(* CODESYS project mobject-datatypes.library
   Company: mobject
   DefaultNamespace: mobject-datatypes
   Version: 0.7.0
   Placeholder: mobject-datatypes
   Author: mobject dev team
   Title: mobject-datatypes

Project tree, tasks and I/O mapping:
  libraries: mobject-collections, 1.2.0 (mobject); mobject-constants-datatype-limits, 1.0.0 (mobject); mobject-deserialization, 0.2.0 (mobject); mobject-disposable, 1.0.0 (mobject); mobject-enumerable, 1.1.0 (mobject); mobject-errors, 0.2.0 (mobject); mobject-events, 1.0.0 (mobject); mobject-serialization, 0.4.0 (mobject); Tc2_Standard, * (Beckhoff Automation GmbH); Tc2_System, * (Beckhoff Automation GmbH); Tc2_Utilities, * (Beckhoff Automation GmbH)
  _Internal/
    Datatype/
      function block DatatypeBase [ST]: OnSerializeTypeWith, Accept, Address, ClearReference, Clone, IsUserDefined, SerializeTypeWith, SerializeWith, Size, TryCopyFrom, TryDeserializeFrom, TryMakeReferenceTo, TryResolveAsAliasDatatype, TryResolveAsEnumDatatype, TryResolveAsInterfaceDatatype, TryResolveAsStructuredDatatype, TypeName
    Errors/
      function block UnknownEnumerationError [ST]: FB_init, ErrorType, Message
    Events/
      function block AliasDatatypeAddedEvent [ST]: FB_init, Target
      function block DatatypeAddedEvent [ST]: FB_init, Target
      function block EnumDatatypeAddedEvent [ST]: FB_init, Target
      function block StructuredDatatypeAddedEvent [ST]: FB_init, Target
    StructureMembers/
      Host/
        function block StructureMemberHost [ST]: Accept, AddMember, GetMemberEnumerator, SerializeTypeWith, SerializeWith, TryDeserializeFrom, TryGetMemberByName
      Interface/
        interface I_HostStructureMembers: Members
        interface I_StructureMembers: Accept, GetMemberEnumerator, TryGetMemberByName
  Datatype/
    Interface/
      interface I_AliasDatatype: BaseDatatype
      interface I_Datatype: Accept, Address, ClearReference, Clone, IsUserDefined, SerializeTypeWith, Size, TryCopyFrom, TryDeserializeFrom, TryMakeReferenceTo, TryResolveAsAliasDatatype, TryResolveAsEnumDatatype, TryResolveAsInterfaceDatatype, TryResolveAsStructuredDatatype, TypeName
      interface I_EnumDatatype
      interface I_InterfaceDatatype: Identifier
      interface I_NumericDatatype: IsFloat, IsSigned
      interface I_StructuredDatatype
      interface I_UserDefinedDatatype: Identifier
    function block AliasDatatypeBase [ST]: AddBaseDatatype, OnSerializeTypeWith, BaseDatatype, SerializeWith, TryDeserializeFrom, TryResolveAsAliasDatatype, TypeName
    function block EnumDatatypeBase [ST]: CreateEnumError, SerializeBaseType, SerializeEnums, AddBaseDatatype, AddEnumeration, IsEnumeratorValueEqual, OnSerializeTypeWith, BaseDatatype, SerializeWith, TryDeserializeFrom, TryResolveAsEnumDatatype, TypeName
    function block InterfaceDatatypeBase [ST]: OnSerializeTypeWith, Identifier, IsUserDefined, TryCopyFrom, TryResolveAsInterfaceDatatype, TypeName
    function block NumericDatatypeBase [ST]: OnSerializeTypeWith, SerializeMaxValue, SerializeMinValue, IsFloat, IsSigned
    function block StructuredDatatypeBase [ST]: AddMember, OnSerializeTypeWith, Accept, Members, SerializeWith, TryDeserializeFrom, TryResolveAsStructuredDatatype, TypeName
    function block UserDefinedDatatypeBase [ST]: OnSerializeTypeWith, Identifier, IsUserDefined, TryCopyFrom
  DatatypeOperations/
    Collection/
      function block DatatypeOperations [ST]: FB_exit, CreateMemoryCopyOperation, CreateSafeMemoryCopyOperation, AddMemoryCopyOperation, AddSafeMemoryCopyOperation, Clear, Execute
    Interface/
      interface I_DatatypeOperation: Execute
    function block MemCopyOperation [ST]: FB_init, Execute
    function block SafeMemCopyOperation [ST]: FB_init, Execute
  DatatypePack/
    interface I_DatatypePack: RegisterWith
  Datatypes/
    Base/
      function block Datatypes [ST]: AcceptAlias, AcceptEnum, AcceptPrimative, AcceptStructures, SerializeAliasTypeWith, SerializeEnumsTypeWith, SerializePrimitiveTypeWith, SerializeStructuresTypeWith, EmitOnAliasDatatypeAddedEvent, EmitOnDatatypeAddedEvent, EmitOnEnumDatatypeAddedEvent, EmitOnStructuredDatatypeAddedEvent, Accept, GetAliasByIdentifier, GetEnumByIdentifier, GetPrimitiveByTypeName, GetStructureByIdentifier, OffEvent, OnceEvent, OnEvent, RegisterDatatype, SerializeTypeWith
    Events/
      interface I_AliasDatatypeAddedEvent: Target
      interface I_DatatypeAddedEvent: Target
      interface I_EnumDatatypeAddedEvent: Target
      interface I_StructuredDatatypeAddedEvent: Target
    Interface/
      interface I_Datatypes: Accept, GetAliasByIdentifier, GetPrimitiveByTypeName, GetStructureByIdentifier, RegisterDatatype, SerializeTypeWith
  DatatypeVisitor/
    interface I_DatatypeVisitor: VisitDatatype
  Primitive/
    function block _BOOL [ST]: FB_init, Address, ClearReference, Clone, MakeReferenceTo, SerializeWith, Size, TryDeserializeFrom, TryMakeReferenceTo, TypeName, Value
    function block _BYTE [ST]: FB_init, SerializeMaxValue, SerializeMinValue, Address, ClearReference, Clone, IsFloat, IsSigned, MakeReferenceTo, MaxValue, MinValue, SerializeWith, Size, TryDeserializeFrom, TryMakeReferenceTo, TypeName, Value
    function block _DINT [ST]: FB_init, SerializeMaxValue, SerializeMinValue, Address, ClearReference, Clone, IsFloat, IsSigned, MakeReferenceTo, MaxValue, MinValue, SerializeWith, Size, TryDeserializeFrom, TryMakeReferenceTo, TypeName, Value
    function block _DT [ST]: FB_init, Address, ClearReference, Clone, MakeReferenceTo, SerializeWith, Size, TryDeserializeFrom, TryMakeReferenceTo, TypeName, Value
    function block _DWORD [ST]: FB_init, SerializeMaxValue, SerializeMinValue, Address, ClearReference, Clone, IsFloat, IsSigned, MakeReferenceTo, MaxValue, MinValue, SerializeWith, Size, TryDeserializeFrom, TryMakeReferenceTo, TypeName, Value
    function block _INT [ST]: FB_init, SerializeMaxValue, SerializeMinValue, Address, ClearReference, Clone, IsFloat, IsSigned, MakeReferenceTo, MaxValue, MinValue, SerializeWith, Size, TryDeserializeFrom, TryMakeReferenceTo, TypeName, Value
    function block _LINT [ST]: FB_init, SerializeMaxValue, SerializeMinValue, Address, ClearReference, Clone, IsFloat, IsSigned, MakeReferenceTo, MaxValue, MinValue, SerializeWith, Size, TryDeserializeFrom, TryMakeReferenceTo, TypeName, Value
    function block _LREAL [ST]: FB_init, SerializeMaxValue, SerializeMinValue, Address, ClearReference, Clone, IsFloat, IsSigned, MakeReferenceTo, MaxValue, MinValue, SerializeWith, Size, TryDeserializeFrom, TryMakeReferenceTo, TypeName, Value
    function block _LWORD [ST]: FB_init, SerializeMaxValue, SerializeMinValue, Address, ClearReference, Clone, IsFloat, IsSigned, MakeReferenceTo, MaxValue, MinValue, SerializeWith, Size, TryDeserializeFrom, TryMakeReferenceTo, TypeName, Value
    function block _REAL [ST]: FB_init, SerializeMaxValue, SerializeMinValue, Address, ClearReference, Clone, IsFloat, IsSigned, MakeReferenceTo, MaxValue, MinValue, SerializeWith, Size, TryDeserializeFrom, TryMakeReferenceTo, TypeName, Value
    function block _SINT [ST]: FB_init, SerializeMaxValue, SerializeMinValue, Address, ClearReference, Clone, IsFloat, IsSigned, MakeReferenceTo, MaxValue, MinValue, SerializeWith, Size, TryDeserializeFrom, TryMakeReferenceTo, TypeName, Value
    function block _STRING [ST]: FB_init, Address, ClearReference, Clone, MakeReferenceTo, SerializeWith, Size, TryDeserializeFrom, TryMakeReferenceTo, TypeName, Value
    function block _TIME_OF_DAY [ST]: FB_init, Address, ClearReference, Clone, MakeReferenceTo, SerializeWith, Size, TryDeserializeFrom, TryMakeReferenceTo, TypeName, Value
    function block _TOD [ST]: FB_init, Address, ClearReference, Clone, MakeReferenceTo, SerializeWith, Size, TryDeserializeFrom, TryMakeReferenceTo, TypeName, Value
    function block _UDINT [ST]: FB_init, SerializeMaxValue, SerializeMinValue, Address, ClearReference, Clone, IsFloat, IsSigned, MakeReferenceTo, MaxValue, MinValue, SerializeWith, Size, TryDeserializeFrom, TryMakeReferenceTo, TypeName, Value
    function block _UINT [ST]: FB_init, SerializeMaxValue, SerializeMinValue, Address, ClearReference, Clone, IsFloat, IsSigned, MakeReferenceTo, MaxValue, MinValue, SerializeWith, Size, TryDeserializeFrom, TryMakeReferenceTo, TypeName, Value
    function block _ULINT [ST]: FB_init, SerializeMaxValue, SerializeMinValue, Address, ClearReference, Clone, IsFloat, IsSigned, MakeReferenceTo, MaxValue, MinValue, SerializeWith, Size, TryDeserializeFrom, TryMakeReferenceTo, TypeName, Value
    function block _USINT [ST]: FB_init, SerializeMaxValue, SerializeMinValue, Address, ClearReference, Clone, IsFloat, IsSigned, MakeReferenceTo, MaxValue, MinValue, SerializeWith, Size, TryDeserializeFrom, TryMakeReferenceTo, TypeName, Value
    function block _WORD [ST]: FB_init, SerializeMaxValue, SerializeMinValue, Address, ClearReference, Clone, IsFloat, IsSigned, MakeReferenceTo, MaxValue, MinValue, SerializeWith, Size, TryDeserializeFrom, TryMakeReferenceTo, TypeName, Value
  function block PrimitiveDatatypePack [ST]: RegisterWith
*)

// _Internal/Datatype/DatatypeBase
{attribute 'linkalways'} 
{attribute 'no_explicit_call' := 'This FB is a CLASS and must be accessed using methods or properties'}
{attribute 'enable_dynamic_creation'}
FUNCTION_BLOCK ABSTRACT DatatypeBase EXTENDS Disposable IMPLEMENTS I_Datatype
VAR
END_VAR

METHOD PROTECTED OnSerializeTypeWith
VAR_INPUT
	Serializer : I_Serializer;
END_VAR
Serializer.AddKeyString('typeName',TypeName);
END_METHOD

METHOD PUBLIC Accept
VAR_INPUT
	Visitor : I_DatatypeVisitor;
END_VAR
Visitor.VisitDatatype(this^);
END_METHOD

PROPERTY PUBLIC ABSTRACT Address : PVOID
GET
END_GET
END_PROPERTY

METHOD PUBLIC ABSTRACT ClearReference
VAR_INPUT
END_VAR
END_METHOD

METHOD PUBLIC ABSTRACT Clone : I_Datatype
END_METHOD

PROPERTY PUBLIC IsUserDefined : BOOL
GET
IsUserDefined := FALSE;
END_GET
END_PROPERTY

METHOD PUBLIC SerializeTypeWith
VAR_INPUT
	Serializer : I_Serializer;
END_VAR
Serializer.StartObject();
OnSerializeTypeWith(Serializer);
Serializer.EndObject();
END_METHOD

METHOD PUBLIC ABSTRACT SerializeWith
VAR_INPUT
	Serializer : I_Serializer;
END_VAR
END_METHOD

PROPERTY PUBLIC ABSTRACT Size : UDINT
GET
END_GET
END_PROPERTY

METHOD PUBLIC TryCopyFrom : BOOL
VAR_INPUT
	Source : I_Datatype;
END_VAR
IF Source.TypeName <> TypeName THEN
	RETURN;
END_IF

memcpy(Address, Source.Address, Size);
TryCopyFrom := TRUE;
END_METHOD

METHOD PUBLIC ABSTRACT TryDeserializeFrom : BOOL
VAR_INPUT
	Deserializer : I_Deserializer;
	Feedback : I_DeserializerFeedback;
END_VAR
END_METHOD

METHOD PUBLIC ABSTRACT TryMakeReferenceTo : BOOL
VAR_INPUT
	Target : I_Datatype;
END_VAR
END_METHOD

METHOD PUBLIC TryResolveAsAliasDatatype : BOOL
VAR_INPUT
	Destination : REFERENCE TO I_AliasDatatype;
END_VAR
TryResolveAsAliasDatatype := FALSE;
END_METHOD

METHOD PUBLIC TryResolveAsEnumDatatype : BOOL
VAR_INPUT
	Destination : REFERENCE TO I_EnumDatatype;
END_VAR
TryResolveAsEnumDatatype := FALSE;
END_METHOD

METHOD PUBLIC TryResolveAsInterfaceDatatype : BOOL
VAR_INPUT
	Destination : REFERENCE TO I_InterfaceDatatype;
END_VAR
TryResolveAsInterfaceDatatype := FALSE;
END_METHOD

METHOD PUBLIC TryResolveAsStructuredDatatype : BOOL
VAR_INPUT
	Destination : REFERENCE TO I_StructuredDatatype;
END_VAR
TryResolveAsStructuredDatatype := FALSE;
END_METHOD

PROPERTY PUBLIC ABSTRACT TypeName : T_MAXSTRING
GET
END_GET
END_PROPERTY

END_FUNCTION_BLOCK

// Datatype/Interface/I_Datatype
INTERFACE I_Datatype extends I_Serializable, I_Deserializable, I_Disposable

METHOD PUBLIC Accept
VAR_INPUT
	Visitor : I_DatatypeVisitor;
END_VAR
END_METHOD

PROPERTY PUBLIC Address : PVOID
GET
END_GET
END_PROPERTY

METHOD PUBLIC ClearReference
VAR_INPUT
END_VAR
END_METHOD

METHOD Clone : I_Datatype
END_METHOD

PROPERTY PUBLIC IsUserDefined : BOOL
GET
END_GET
END_PROPERTY

METHOD PUBLIC SerializeTypeWith
VAR_INPUT
	Serializer : I_Serializer;
END_VAR
END_METHOD

PROPERTY PUBLIC Size : UDINT
GET
END_GET
END_PROPERTY

METHOD PUBLIC TryCopyFrom : BOOL
VAR_INPUT
	Source : I_Datatype;
END_VAR
END_METHOD

METHOD PUBLIC ABSTRACT TryDeserializeFrom : BOOL
VAR_INPUT
	Deserializer : I_Deserializer;
	Feedback : I_DeserializerFeedback;
END_VAR
END_METHOD

METHOD TryMakeReferenceTo : BOOL
VAR_INPUT
	Target : I_Datatype;
END_VAR
END_METHOD

METHOD PUBLIC TryResolveAsAliasDatatype : BOOL
VAR_INPUT
	Destination : REFERENCE TO I_AliasDatatype;
END_VAR
END_METHOD

METHOD PUBLIC TryResolveAsEnumDatatype : BOOL
VAR_INPUT
	Destination : REFERENCE TO I_EnumDatatype;
END_VAR
END_METHOD

METHOD PUBLIC TryResolveAsInterfaceDatatype : BOOL
VAR_INPUT
	Destination : REFERENCE TO I_InterfaceDatatype;
END_VAR
END_METHOD

METHOD PUBLIC TryResolveAsStructuredDatatype : BOOL
VAR_INPUT
	Destination : REFERENCE TO I_StructuredDatatype;
END_VAR
END_METHOD

PROPERTY PUBLIC TypeName : T_MAXSTRING
GET
END_GET
END_PROPERTY

END_INTERFACE

// DatatypeVisitor/I_DatatypeVisitor
INTERFACE I_DatatypeVisitor

METHOD VisitDatatype
VAR_INPUT
	VisitingDatatype : I_Datatype;
END_VAR
END_METHOD

END_INTERFACE

// Datatype/Interface/I_AliasDatatype
INTERFACE I_AliasDatatype EXTENDS I_UserDefinedDatatype

PROPERTY PUBLIC BaseDatatype : I_Datatype
GET
END_GET
END_PROPERTY

END_INTERFACE

// Datatype/Interface/I_UserDefinedDatatype
INTERFACE I_UserDefinedDatatype EXTENDS I_Datatype

PROPERTY PUBLIC Identifier : T_MAXSTRING
GET
END_GET
END_PROPERTY

END_INTERFACE

// Datatype/Interface/I_EnumDatatype
INTERFACE I_EnumDatatype EXTENDS I_UserDefinedDatatype

END_INTERFACE

// Datatype/Interface/I_InterfaceDatatype
INTERFACE I_InterfaceDatatype EXTENDS I_Datatype

PROPERTY PUBLIC Identifier : T_MAXSTRING
GET
END_GET
END_PROPERTY

END_INTERFACE

// Datatype/Interface/I_StructuredDatatype
INTERFACE I_StructuredDatatype EXTENDS I_UserDefinedDatatype, I_HostStructureMembers

END_INTERFACE

// _Internal/StructureMembers/Interface/I_HostStructureMembers
INTERFACE I_HostStructureMembers EXTENDS __SYSTEM.IQueryInterface

PROPERTY PUBLIC Members : I_StructureMembers
GET
END_GET
END_PROPERTY

END_INTERFACE

// _Internal/StructureMembers/Interface/I_StructureMembers
INTERFACE I_StructureMembers

METHOD PUBLIC Accept
VAR_INPUT
	Visitor : I_DatatypeVisitor;
END_VAR
END_METHOD

METHOD PUBLIC GetMemberEnumerator : I_KeyValueForwardEnumerator
VAR_INPUT
END_VAR
END_METHOD

METHOD PUBLIC TryGetMemberByName : BOOL
VAR_INPUT
	Name : T_MAXSTRING;
	Destination : REFERENCE TO I_Datatype;
END_VAR
END_METHOD

END_INTERFACE

// _Internal/Errors/UnknownEnumerationError
{attribute 'linkalways'} 
{attribute 'no_explicit_call' := 'This FB is a CLASS and must be accessed using methods or properties'}
{attribute 'enable_dynamic_creation'}
FUNCTION_BLOCK UnknownEnumerationError EXTENDS Error
VAR
	enumString : T_MAXSTRING;
END_VAR

METHOD FB_init : BOOL
VAR_INPUT
	bInitRetains : BOOL; // if TRUE, the retain variables are initialized (warm start / cold start)
	bInCopyCode : BOOL;  // if TRUE, the instance afterwards gets moved into the copy code (online change)
	EnumString : T_MAXSTRING;
END_VAR
THIS^.enumString := EnumString;
END_METHOD

PROPERTY PUBLIC ErrorType : T_MAXSTRING
GET
ErrorType := 'UNKNOWN_ENUMERATION_ERROR';
END_GET
END_PROPERTY

PROPERTY PUBLIC Message : T_MAXSTRING
GET
Message := CONCAT('Unknown Enumeration : ', enumString);
END_GET
END_PROPERTY

END_FUNCTION_BLOCK

// _Internal/Events/AliasDatatypeAddedEvent
{attribute 'linkalways'} 
{attribute 'no_explicit_call' := 'This FB is a CLASS and must be accessed using methods or properties'}
{attribute 'enable_dynamic_creation'}
FUNCTION_BLOCK AliasDatatypeAddedEvent EXTENDS Disposable IMPLEMENTS I_AliasDatatypeAddedEvent
VAR
	_target : I_AliasDatatype;
END_VAR

METHOD FB_init : BOOL
VAR_INPUT
	bInitRetains : BOOL; // if TRUE, the retain variables are initialized (warm start / cold start)
	bInCopyCode : BOOL;  // if TRUE, the instance afterwards gets moved into the copy code (online change)
	Target : I_AliasDatatype;
END_VAR
This^._target := Target;
END_METHOD

PROPERTY PUBLIC Target : I_AliasDatatype
GET
Target := _target;
END_GET
END_PROPERTY

END_FUNCTION_BLOCK

// Datatypes/Events/I_AliasDatatypeAddedEvent
INTERFACE I_AliasDatatypeAddedEvent EXTENDS I_Event

PROPERTY PUBLIC Target : I_AliasDatatype
GET
END_GET
END_PROPERTY

END_INTERFACE

// _Internal/Events/DatatypeAddedEvent
{attribute 'linkalways'} 
{attribute 'no_explicit_call' := 'This FB is a CLASS and must be accessed using methods or properties'}
{attribute 'enable_dynamic_creation'}
FUNCTION_BLOCK DatatypeAddedEvent EXTENDS Disposable IMPLEMENTS I_DatatypeAddedEvent
VAR
	_target : I_Datatype;
END_VAR

METHOD FB_init : BOOL
VAR_INPUT
	bInitRetains : BOOL; // if TRUE, the retain variables are initialized (warm start / cold start)
	bInCopyCode : BOOL;  // if TRUE, the instance afterwards gets moved into the copy code (online change)
	Target : I_Datatype;
END_VAR
This^._target := Target;
END_METHOD

PROPERTY PUBLIC Target : I_Datatype
GET
Target := _target;
END_GET
END_PROPERTY

END_FUNCTION_BLOCK

// Datatypes/Events/I_DatatypeAddedEvent
INTERFACE I_DatatypeAddedEvent EXTENDS I_Event

PROPERTY PUBLIC Target : I_Datatype
GET
END_GET
END_PROPERTY

END_INTERFACE

// _Internal/Events/EnumDatatypeAddedEvent
{attribute 'linkalways'} 
{attribute 'no_explicit_call' := 'This FB is a CLASS and must be accessed using methods or properties'}
{attribute 'enable_dynamic_creation'}
FUNCTION_BLOCK EnumDatatypeAddedEvent EXTENDS Disposable IMPLEMENTS I_EnumDatatypeAddedEvent
VAR
	_target : I_EnumDatatype;
END_VAR

METHOD FB_init : BOOL
VAR_INPUT
	bInitRetains : BOOL; // if TRUE, the retain variables are initialized (warm start / cold start)
	bInCopyCode : BOOL;  // if TRUE, the instance afterwards gets moved into the copy code (online change)
	Target : I_EnumDatatype;
END_VAR
This^._target := Target;
END_METHOD

PROPERTY PUBLIC Target : I_EnumDatatype
GET
Target := _target;
END_GET
END_PROPERTY

END_FUNCTION_BLOCK

// Datatypes/Events/I_EnumDatatypeAddedEvent
INTERFACE I_EnumDatatypeAddedEvent EXTENDS I_Event

PROPERTY PUBLIC Target : I_EnumDatatype
GET
END_GET
END_PROPERTY

END_INTERFACE

// _Internal/Events/StructuredDatatypeAddedEvent
{attribute 'linkalways'} 
{attribute 'no_explicit_call' := 'This FB is a CLASS and must be accessed using methods or properties'}
{attribute 'enable_dynamic_creation'}
FUNCTION_BLOCK StructuredDatatypeAddedEvent EXTENDS Disposable IMPLEMENTS I_StructuredDatatypeAddedEvent
VAR
	_target : I_StructuredDatatype;
END_VAR

METHOD FB_init : BOOL
VAR_INPUT
	bInitRetains : BOOL; // if TRUE, the retain variables are initialized (warm start / cold start)
	bInCopyCode : BOOL;  // if TRUE, the instance afterwards gets moved into the copy code (online change)
	Target : I_StructuredDatatype;
END_VAR
This^._target := Target;
END_METHOD

PROPERTY PUBLIC Target : I_StructuredDatatype
GET
Target := _target;
END_GET
END_PROPERTY

END_FUNCTION_BLOCK

// Datatypes/Events/I_StructuredDatatypeAddedEvent
INTERFACE I_StructuredDatatypeAddedEvent EXTENDS I_Event

PROPERTY PUBLIC Target : I_StructuredDatatype
GET
END_GET
END_PROPERTY

END_INTERFACE

// _Internal/StructureMembers/Host/StructureMemberHost
{attribute 'linkalways'} 
{attribute 'no_explicit_call' := 'This FB is a CLASS and must be accessed using methods or properties'}
{attribute 'enable_dynamic_creation'}
FUNCTION_BLOCK StructureMemberHost IMPLEMENTS I_Serializable, I_StructureMembers
VAR
	members : OrderedDictionary;
END_VAR

METHOD PUBLIC Accept
VAR_INPUT
	Visitor : I_DatatypeVisitor;
END_VAR
VAR
	enumerator : I_ForwardEnumerator;
	member : I_Datatype;
END_VAR
enumerator := members.GetEnumerator();

WHILE (enumerator.MoveNext()) DO
	
	IF enumerator.TryGet(member) THEN
		member.Accept(Visitor);
	END_IF

END_WHILE

enumerator.Dispose();
END_METHOD

METHOD PUBLIC AddMember
VAR_INPUT
	MemberName : T_MAXSTRING;
	Member : I_Datatype;
END_VAR
members.AddOrUpdate(MemberName, Member);
END_METHOD

METHOD PUBLIC GetMemberEnumerator : I_KeyValueForwardEnumerator
VAR_INPUT
END_VAR
GetMemberEnumerator := members.GetKeyValueEnumerator();
END_METHOD

METHOD PUBLIC SerializeTypeWith
VAR_INPUT
	Serializer : I_Serializer;
END_VAR
VAR
	enumerator : I_KeyValueForwardEnumerator;
	member : I_Datatype;
END_VAR
IF members.Count = 0 THEN
	RETURN;
END_IF

Serializer.AddKey('members');
Serializer.StartObject();

enumerator := members.GetKeyValueEnumerator();

WHILE enumerator.MoveNext() DO
	IF enumerator.TryGet(member) THEN
		Serializer.AddKey(enumerator.Key);
		member.SerializeTypeWith(Serializer);
	END_IF
END_WHILE

enumerator.Dispose();

Serializer.EndObject();
END_METHOD

METHOD PUBLIC SerializeWith
VAR_INPUT
	Serializer : I_Serializer;
END_VAR
VAR
	enumerator : I_KeyValueForwardEnumerator;
	member : I_Datatype;
END_VAR
enumerator := members.GetKeyValueEnumerator();

WHILE enumerator.MoveNext() DO
	IF enumerator.TryGet(member) THEN
		Serializer.AddKey(enumerator.Key);
		member.SerializeWith(Serializer);
	END_IF
END_WHILE

enumerator.Dispose();
END_METHOD

METHOD PUBLIC TryDeserializeFrom : BOOL
VAR_INPUT
	Deserializer : I_Deserializer;
	Feedback : I_DeserializerFeedback;
END_VAR
VAR
	membersEnumerator : I_DeserializerObjectForwardEnumerator;
	member : I_Datatype;
END_VAR
membersEnumerator := Deserializer.GetObjectEnumerator();

WHILE membersEnumerator.MoveNext() DO
	
	IF NOT TryGetMemberByName(membersEnumerator.Key, member) THEN
		CONTINUE;
	END_IF
	
	IF NOT member.TryDeserializeFrom(membersEnumerator.Current, Feedback) THEN
		RETURN;
	END_IF

END_WHILE

membersEnumerator.Dispose();
TryDeserializeFrom := TRUE;
END_METHOD

METHOD PUBLIC TryGetMemberByName : BOOL
VAR_INPUT
	Name : T_MAXSTRING;
	Destination : REFERENCE TO I_Datatype;
END_VAR
VAR
	member : I_Datatype;
END_VAR
IF NOT members.TryGetValue(Name, member) THEN
	RETURN;
END_IF

Destination := member;
TryGetMemberByName := TRUE;
END_METHOD

END_FUNCTION_BLOCK

// Datatype/Interface/I_NumericDatatype
INTERFACE I_NumericDatatype EXTENDS I_Datatype

PROPERTY PUBLIC ABSTRACT IsFloat : BOOL
GET
END_GET
END_PROPERTY

PROPERTY PUBLIC IsSigned : BOOL
GET
END_GET
END_PROPERTY

END_INTERFACE

// Datatype/AliasDatatypeBase
{attribute 'linkalways'} 
{attribute 'no_explicit_call' := 'This FB is a CLASS and must be accessed using methods or properties'}
{attribute 'enable_dynamic_creation'}
FUNCTION_BLOCK ABSTRACT AliasDatatypeBase EXTENDS UserDefinedDatatypeBase IMPLEMENTS I_AliasDatatype
VAR
	_baseDatatype : I_Datatype;
END_VAR

METHOD PROTECTED AddBaseDatatype
VAR_INPUT
	BaseType : I_Datatype;
END_VAR
_baseDatatype := BaseType;
END_METHOD

METHOD PROTECTED OnSerializeTypeWith
VAR_INPUT
	Serializer : I_Serializer;
END_VAR
SUPER^.OnSerializeTypeWith(Serializer);
Serializer.AddKey('baseDatatype');
_baseDatatype.SerializeTypeWith(Serializer);
END_METHOD

PROPERTY PUBLIC BaseDatatype : I_Datatype
GET
BaseDatatype := _baseDatatype;
END_GET
END_PROPERTY

METHOD PUBLIC SerializeWith
VAR_INPUT
	Serializer : I_Serializer;
END_VAR
_baseDatatype.SerializeWith(Serializer);
END_METHOD

METHOD TryDeserializeFrom : BOOL
VAR_INPUT
	Deserializer : I_Deserializer;
	Feedback : I_DeserializerFeedback;
END_VAR
TryDeserializeFrom := _baseDatatype.TryDeserializeFrom(Deserializer, Feedback);
END_METHOD

METHOD PUBLIC TryResolveAsAliasDatatype : BOOL
VAR_INPUT
	Destination : REFERENCE TO I_AliasDatatype;
END_VAR
Destination := THIS^;
TryResolveAsAliasDatatype := TRUE;
END_METHOD

PROPERTY PUBLIC TypeName : T_MAXSTRING
GET
TypeName := 'ALIAS';
END_GET
END_PROPERTY

END_FUNCTION_BLOCK

// Datatype/UserDefinedDatatypeBase
{attribute 'linkalways'} 
{attribute 'no_explicit_call' := 'This FB is a CLASS and must be accessed using methods or properties'}
{attribute 'enable_dynamic_creation'}
FUNCTION_BLOCK ABSTRACT UserDefinedDatatypeBase EXTENDS DatatypeBase IMPLEMENTS I_UserDefinedDatatype
VAR
END_VAR

METHOD PROTECTED OnSerializeTypeWith
VAR_INPUT
	Serializer : I_Serializer;
END_VAR
SUPER^.OnSerializeTypeWith(Serializer);
Serializer.AddKeyString('identifier',Identifier);
END_METHOD

PROPERTY PUBLIC ABSTRACT Identifier : T_MAXSTRING
GET
END_GET
END_PROPERTY

PROPERTY PUBLIC IsUserDefined : BOOL
GET
IsUserDefined := TRUE;
END_GET
END_PROPERTY

METHOD PUBLIC TryCopyFrom : BOOL
VAR_INPUT
	Source : I_Datatype;
END_VAR
VAR
	sourceAsUdt : I_UserDefinedDatatype;
END_VAR
IF NOT __QUERYINTERFACE(Source, sourceAsUdt) THEN
	RETURN;
END_IF

IF sourceAsUdt.Identifier <> Identifier THEN
	RETURN;
END_IF

TryCopyFrom := SUPER^.TryCopyFrom(Source);
END_METHOD

END_FUNCTION_BLOCK

// Datatype/EnumDatatypeBase
{attribute 'linkalways'} 
{attribute 'no_explicit_call' := 'This FB is a CLASS and must be accessed using methods or properties'}
{attribute 'enable_dynamic_creation'}
FUNCTION_BLOCK ABSTRACT EnumDatatypeBase EXTENDS UserDefinedDatatypeBase IMPLEMENTS I_EnumDatatype
VAR
	_baseDatatype : I_Datatype;
	enumerations : OrderedDictionary;
END_VAR

METHOD PRIVATE CreateEnumError : I_Error
VAR_INPUT
	Enum : T_MAXSTRING;
END_VAR
VAR
	pError : POINTER TO UnknownEnumerationError;
END_VAR
pError := __NEW(UnknownEnumerationError(EnumString := Enum));
CreateEnumError := pError^;
END_METHOD

METHOD PRIVATE SerializeBaseType
VAR_INPUT
	Serializer : I_Serializer;
END_VAR
IF _baseDatatype = 0 THEN
	RETURN;
END_IF

Serializer.AddKey('baseType');
_baseDatatype.SerializeTypeWith(Serializer);
END_METHOD

METHOD PRIVATE SerializeEnums
VAR_INPUT
	Serializer : I_Serializer;
END_VAR
VAR
	enumerator : I_KeyValueForwardEnumerator;
END_VAR
Serializer.AddKey('enumerations');
Serializer.StartArray();

enumerator := enumerations.GetKeyValueEnumerator();

WHILE enumerator.MoveNext() DO
	Serializer.AddString(enumerator.Key);
END_WHILE

enumerator.Dispose();

Serializer.EndArray();
END_METHOD

METHOD PROTECTED AddBaseDatatype
VAR_INPUT
	BaseType : I_Datatype;
END_VAR
_baseDatatype := BaseType;
END_METHOD

METHOD PROTECTED AddEnumeration
VAR_INPUT
	Enumeration : T_MAXSTRING;
	Value : ANY;
END_VAR
enumerations.AddOrUpdate(Enumeration, Value);
END_METHOD

METHOD ABSTRACT IsEnumeratorValueEqual : BOOL
VAR_INPUT
	Enumerator : I_KeyValueForwardEnumerator;
END_VAR
END_METHOD

METHOD PROTECTED OnSerializeTypeWith
VAR_INPUT
	Serializer : I_Serializer;
END_VAR
SUPER^.OnSerializeTypeWith(Serializer);
SerializeEnums(Serializer);
SerializeBaseType(Serializer);
END_METHOD

PROPERTY PUBLIC BaseDatatype : I_Datatype
GET
BaseDatatype := _baseDatatype;
END_GET
END_PROPERTY

METHOD PUBLIC SerializeWith
VAR_INPUT
	Serializer : I_Serializer;
END_VAR
VAR
	returnKey : T_MAXSTRING;
	enumerator : I_KeyValueForwardEnumerator;
END_VAR
enumerator := enumerations.GetKeyValueEnumerator();
returnKey := 'UNDEFINED';

WHILE (enumerator.MoveNext()) DO
	
	IF IsEnumeratorValueEqual(enumerator) THEN
		returnKey := enumerator.key;
		EXIT;
	END_IF

END_WHILE

Serializer.AddString(returnKey);
enumerator.Dispose();
END_METHOD

METHOD TryDeserializeFrom : BOOL
VAR_INPUT
	Deserializer : I_Deserializer;
	Feedback : I_DeserializerFeedback;
END_VAR
VAR
	key : T_MAXSTRING;
	error : I_Error;
END_VAR
IF NOT Deserializer.TryGetString(key, Feedback) THEN
	RETURN;
END_IF

IF NOT enumerations.TryGetValueTo(key, Address, Size) THEN
	error := CreateEnumError(key);
	Feedback.LogError(error);
	RETURN;
END_IF

TryDeserializeFrom := TRUE;
END_METHOD

METHOD PUBLIC TryResolveAsEnumDatatype : BOOL
VAR_INPUT
	Destination : REFERENCE TO I_EnumDatatype;
END_VAR
Destination := THIS^;
TryResolveAsEnumDatatype := TRUE;
END_METHOD

PROPERTY PUBLIC TypeName : T_MAXSTRING
GET
TypeName := 'ENUM';
END_GET
END_PROPERTY

END_FUNCTION_BLOCK

// Datatype/InterfaceDatatypeBase
{attribute 'linkalways'} 
{attribute 'no_explicit_call' := 'This FB is a CLASS and must be accessed using methods or properties'}
{attribute 'enable_dynamic_creation'}
FUNCTION_BLOCK ABSTRACT InterfaceDatatypeBase EXTENDS DatatypeBase IMPLEMENTS I_InterfaceDatatype
VAR
END_VAR

METHOD PROTECTED OnSerializeTypeWith
VAR_INPUT
	Serializer : I_Serializer;
END_VAR
SUPER^.OnSerializeTypeWith(Serializer);
Serializer.AddKeyString('identifier',Identifier);
END_METHOD

PROPERTY PUBLIC ABSTRACT Identifier : T_MAXSTRING
GET
END_GET
END_PROPERTY

PROPERTY PUBLIC IsUserDefined : BOOL
GET
IsUserDefined := FALSE;
END_GET
END_PROPERTY

METHOD PUBLIC TryCopyFrom : BOOL
VAR_INPUT
	Source : I_Datatype;
END_VAR
VAR
	sourceAsInterface : I_InterfaceDatatype;
END_VAR
IF NOT __QUERYINTERFACE(Source, sourceAsInterface) THEN
	RETURN;
END_IF

IF sourceAsInterface.Identifier <> Identifier THEN
	RETURN;
END_IF

TryCopyFrom := SUPER^.TryCopyFrom(Source);
END_METHOD

METHOD PUBLIC TryResolveAsInterfaceDatatype : BOOL
VAR_INPUT
	Destination : REFERENCE TO I_InterfaceDatatype;
END_VAR
Destination := THIS^;
TryResolveAsInterfaceDatatype := TRUE;
END_METHOD

PROPERTY PUBLIC TypeName : T_MAXSTRING
GET
TypeName := 'INTERFACE';
END_GET
END_PROPERTY

END_FUNCTION_BLOCK

// Datatype/NumericDatatypeBase
{attribute 'linkalways'} 
{attribute 'no_explicit_call' := 'This FB is a CLASS and must be accessed using methods or properties'}
{attribute 'enable_dynamic_creation'}
FUNCTION_BLOCK ABSTRACT NumericDatatypeBase EXTENDS DatatypeBase IMPLEMENTS I_NumericDatatype
VAR
END_VAR

METHOD PROTECTED OnSerializeTypeWith
VAR_INPUT
	Serializer : I_Serializer;
END_VAR
SUPER^.OnSerializeTypeWith(Serializer);
Serializer.AddKey('minValue');
SerializeMinValue(Serializer);
Serializer.AddKey('maxValue');
SerializeMaxValue(Serializer);
Serializer.AddKeyBool('isSigned', IsSigned);
Serializer.AddKeyBool('isFloat', IsFloat);
END_METHOD

METHOD PROTECTED ABSTRACT SerializeMaxValue
VAR_INPUT
	Serializer : I_Serializer;
END_VAR
END_METHOD

METHOD PROTECTED ABSTRACT SerializeMinValue
VAR_INPUT
	Serializer : I_Serializer;
END_VAR
END_METHOD

PROPERTY PUBLIC ABSTRACT IsFloat : BOOL
GET
END_GET
END_PROPERTY

PROPERTY PUBLIC ABSTRACT IsSigned : BOOL
GET
END_GET
END_PROPERTY

END_FUNCTION_BLOCK

// Datatype/StructuredDatatypeBase
{attribute 'linkalways'} 
{attribute 'no_explicit_call' := 'This FB is a CLASS and must be accessed using methods or properties'}
{attribute 'enable_dynamic_creation'}
FUNCTION_BLOCK ABSTRACT StructuredDatatypeBase EXTENDS UserDefinedDatatypeBase IMPLEMENTS I_StructuredDatatype
VAR
	membersHost : StructureMemberHost;
END_VAR

METHOD PROTECTED AddMember
VAR_INPUT
	MemberName : T_MAXSTRING;
	Member : I_Datatype;
END_VAR
membersHost.AddMember(MemberName, Member);
END_METHOD

METHOD PROTECTED OnSerializeTypeWith
VAR_INPUT
	Serializer : I_Serializer;
END_VAR
SUPER^.OnSerializeTypeWith(Serializer);
membersHost.SerializeTypeWith(Serializer);
END_METHOD

METHOD PUBLIC Accept
VAR_INPUT
	Visitor : I_DatatypeVisitor;
END_VAR
Visitor.VisitDatatype(THIS^);
membersHost.Accept(Visitor);
END_METHOD

PROPERTY PUBLIC Members : I_StructureMembers
GET
Members := membersHost;
END_GET
END_PROPERTY

METHOD PUBLIC SerializeWith
VAR_INPUT
	Serializer : I_Serializer;
END_VAR
Serializer.StartObject();
membersHost.SerializeWith(Serializer);
Serializer.EndObject();
END_METHOD

METHOD TryDeserializeFrom : BOOL
VAR_INPUT
	Deserializer : I_Deserializer;
	Feedback : I_DeserializerFeedback;
END_VAR
TryDeserializeFrom := membersHost.TryDeserializeFrom(Deserializer, Feedback);
END_METHOD

METHOD PUBLIC TryResolveAsStructuredDatatype : BOOL
VAR_INPUT
	Destination : REFERENCE TO I_StructuredDatatype;
END_VAR
Destination := THIS^;
TryResolveAsStructuredDatatype := TRUE;
END_METHOD

PROPERTY PUBLIC TypeName : T_MAXSTRING
GET
TypeName := 'STRUCT';
END_GET
END_PROPERTY

END_FUNCTION_BLOCK

// DatatypeOperations/Collection/DatatypeOperations
{attribute 'linkalways'} 
{attribute 'no_explicit_call' := 'This FB is a CLASS and must be accessed using methods or properties'}
{attribute 'enable_dynamic_creation'}
FUNCTION_BLOCK DatatypeOperations
VAR
	operations : Stack;
END_VAR

METHOD FB_exit : BOOL
VAR_INPUT
	bInCopyCode : BOOL; // if TRUE, the exit method is called for exiting an instance that is copied afterwards (online change).
END_VAR
IF bInCopyCode THEN
	RETURN;
END_IF

operations.Clear();
END_METHOD

METHOD PRIVATE CreateMemoryCopyOperation : I_DatatypeOperation
VAR_INPUT
	OperationSource : I_Datatype;
	OperationDestination : I_Datatype;
END_VAR
VAR
	pOperation : POINTER TO MemCopyOperation;
END_VAR
pOperation := __NEW(MemCopyOperation(Source := OperationSource, Destination := OperationDestination));
CreateMemoryCopyOperation := pOperation^;
END_METHOD

METHOD PRIVATE CreateSafeMemoryCopyOperation : I_DatatypeOperation
VAR_INPUT
	OperationSource : I_Datatype;
	OperationDestination : I_Datatype;
END_VAR
VAR
	pOperation : POINTER TO SafeMemCopyOperation;
END_VAR
pOperation := __NEW(SafeMemCopyOperation(Source := OperationSource, Destination := OperationDestination));
CreateSafeMemoryCopyOperation := pOperation^;
END_METHOD

METHOD PUBLIC AddMemoryCopyOperation
VAR_INPUT
	Source : I_Datatype;
	Destination : I_Datatype;
END_VAR
VAR
	operation : I_DatatypeOperation;
END_VAR
operation := CreateMemoryCopyOperation(Source,Destination);
operations.Push(operation);
END_METHOD

METHOD PUBLIC AddSafeMemoryCopyOperation
VAR_INPUT
	Source : I_Datatype;
	Destination : I_Datatype;
END_VAR
VAR
	operation : I_DatatypeOperation;
END_VAR
operation := CreateSafeMemoryCopyOperation(Source,Destination);
operations.Push(operation);
END_METHOD

METHOD PUBLIC Clear
VAR
	operation : I_DatatypeOperation;
END_VAR
WHILE operations.TryPop(operation) DO
	operation.Dispose();
END_WHILE
END_METHOD

METHOD PUBLIC Execute
VAR
	enumerator : I_ForwardEnumerator;
	operation : I_DatatypeOperation;
END_VAR
enumerator := operations.GetEnumerator();

WHILE enumerator.MoveNext() DO
	IF enumerator.TryGet(operation) THEN
		operation.Execute();
	END_IF
END_WHILE

enumerator.Dispose();
END_METHOD

END_FUNCTION_BLOCK

// DatatypeOperations/MemCopyOperation
{attribute 'linkalways'} 
{attribute 'no_explicit_call' := 'This FB is a CLASS and must be accessed using methods or properties'}
{attribute 'enable_dynamic_creation'}
FUNCTION_BLOCK MemCopyOperation EXTENDS Disposable IMPLEMENTS I_DatatypeOperation
VAR
	source : I_Datatype;
	destination : I_Datatype;
END_VAR

METHOD FB_init : BOOL
VAR_INPUT
	bInitRetains : BOOL; // if TRUE, the retain variables are initialized (warm start / cold start)
	bInCopyCode : BOOL;  // if TRUE, the instance afterwards gets moved into the copy code (online change)
	Source : I_Datatype;
	Destination : I_Datatype;
END_VAR
THIS^.source := Source;
This^.destination := Destination;
END_METHOD

METHOD Execute
VAR
END_VAR
memcpy(destination.Address, source.Address, source.Size);
END_METHOD

END_FUNCTION_BLOCK

// DatatypeOperations/Interface/I_DatatypeOperation
INTERFACE I_DatatypeOperation EXTENDS I_Disposable

METHOD Execute
VAR
END_VAR
END_METHOD

END_INTERFACE

// DatatypeOperations/SafeMemCopyOperation
{attribute 'linkalways'} 
{attribute 'no_explicit_call' := 'This FB is a CLASS and must be accessed using methods or properties'}
{attribute 'enable_dynamic_creation'}
FUNCTION_BLOCK SafeMemCopyOperation EXTENDS Disposable IMPLEMENTS I_DatatypeOperation
VAR
	source : I_Datatype;
	destination : I_Datatype;
END_VAR

METHOD FB_init : BOOL
VAR_INPUT
	bInitRetains : BOOL; // if TRUE, the retain variables are initialized (warm start / cold start)
	bInCopyCode : BOOL;  // if TRUE, the instance afterwards gets moved into the copy code (online change)
	Source : I_Datatype;
	Destination : I_Datatype;
END_VAR
THIS^.source := Source;
This^.destination := Destination;
END_METHOD

METHOD Execute
VAR
END_VAR
destination.TryCopyFrom(source);
END_METHOD

END_FUNCTION_BLOCK

// DatatypePack/I_DatatypePack
INTERFACE I_DatatypePack

METHOD RegisterWith
VAR_INPUT
	Datatypes : I_Datatypes;
END_VAR
END_METHOD

END_INTERFACE

// Datatypes/Base/Datatypes
{attribute 'linkalways'} 
{attribute 'no_explicit_call' := 'This FB is a CLASS and must be accessed using methods or properties'}
{attribute 'enable_dynamic_creation'}
FUNCTION_BLOCK Datatypes IMPLEMENTS I_Datatypes
VAR
	eventEmitter : EventEmitter;
	primitives : OrderedDictionary;
	structures : OrderedDictionary;
	alias : OrderedDictionary;
	enums : OrderedDictionary;
END_VAR

METHOD PRIVATE AcceptAlias
VAR_INPUT
	Visitor : I_DatatypeVisitor;
END_VAR
VAR
	enumerator : I_ForwardEnumerator;
	datatype : I_AliasDatatype;
END_VAR
enumerator := alias.GetEnumerator();

WHILE enumerator.MoveNext() DO
	IF enumerator.TryGet(datatype) THEN
		datatype.Accept(Visitor);
	END_IF
END_WHILE

enumerator.Dispose();
END_METHOD

METHOD PRIVATE AcceptEnum
VAR_INPUT
	Visitor : I_DatatypeVisitor;
END_VAR
VAR
	enumerator : I_ForwardEnumerator;
	datatype : I_EnumDatatype;
END_VAR
enumerator := enums.GetEnumerator();

WHILE enumerator.MoveNext() DO
	IF enumerator.TryGet(datatype) THEN
		datatype.Accept(Visitor);
	END_IF
END_WHILE

enumerator.Dispose();
END_METHOD

METHOD PRIVATE AcceptPrimative
VAR_INPUT
	Visitor : I_DatatypeVisitor;
END_VAR
VAR
	enumerator : I_ForwardEnumerator;
	datatype : I_Datatype;
END_VAR
enumerator := primitives.GetEnumerator();

WHILE enumerator.MoveNext() DO
	IF enumerator.TryGet(datatype) THEN
		datatype.Accept(Visitor);
	END_IF
END_WHILE

enumerator.Dispose();
END_METHOD

METHOD PRIVATE AcceptStructures
VAR_INPUT
	Visitor : I_DatatypeVisitor;
END_VAR
VAR
	enumerator : I_ForwardEnumerator;
	datatype : I_StructuredDatatype;
END_VAR
enumerator := structures.GetEnumerator();

WHILE enumerator.MoveNext() DO	
	IF enumerator.TryGet(datatype) THEN
		datatype.Accept(Visitor);
	END_IF
END_WHILE

enumerator.Dispose();
END_METHOD

METHOD PRIVATE SerializeAliasTypeWith
VAR_INPUT
	Serializer : I_Serializer;
END_VAR
VAR
	enumerator : I_ForwardEnumerator;
	datatype : I_AliasDatatype;
END_VAR
enumerator := alias.GetEnumerator();

WHILE enumerator.MoveNext() DO
	IF enumerator.TryGet(datatype) THEN
		datatype.SerializeTypeWith(Serializer);
	END_IF
END_WHILE

enumerator.Dispose();
END_METHOD

METHOD PRIVATE SerializeEnumsTypeWith
VAR_INPUT
	Serializer : I_Serializer;
END_VAR
VAR
	enumerator : I_ForwardEnumerator;
	datatype : I_EnumDatatype;
END_VAR
enumerator := enums.GetEnumerator();

WHILE enumerator.MoveNext() DO
	IF enumerator.TryGet(datatype) THEN
		datatype.SerializeTypeWith(Serializer);
	END_IF
END_WHILE

enumerator.Dispose();
END_METHOD

METHOD PRIVATE SerializePrimitiveTypeWith
VAR_INPUT
	Serializer : I_Serializer;
END_VAR
VAR
	enumerator : I_ForwardEnumerator;
	datatype : I_Datatype;
END_VAR
enumerator := primitives.GetEnumerator();

WHILE enumerator.MoveNext() DO
	IF enumerator.TryGet(datatype) THEN
		datatype.SerializeTypeWith(Serializer);
	END_IF
END_WHILE

enumerator.Dispose();
END_METHOD

METHOD PRIVATE SerializeStructuresTypeWith
VAR_INPUT
	Serializer : I_Serializer;
END_VAR
VAR
	enumerator : I_ForwardEnumerator;
	datatype : I_StructuredDatatype;
END_VAR
enumerator := structures.GetEnumerator();

WHILE enumerator.MoveNext() DO
	IF enumerator.TryGet(datatype) THEN
		datatype.SerializeTypeWith(Serializer);
	END_IF
END_WHILE

enumerator.Dispose();
END_METHOD

METHOD PROTECTED EmitOnAliasDatatypeAddedEvent
VAR_INPUT
	Datatype : I_AliasDatatype;
END_VAR
VAR
	pAliasDatatypeAddedEvent : POINTER TO AliasDatatypeAddedEvent;
END_VAR
pAliasDatatypeAddedEvent := __NEW(AliasDatatypeAddedEvent(Target := Datatype));
eventEmitter.Emit('OnDatatypeAdded',pAliasDatatypeAddedEvent^);
pAliasDatatypeAddedEvent^.Dispose();
END_METHOD

METHOD PROTECTED EmitOnDatatypeAddedEvent
VAR_INPUT
	Datatype : I_Datatype;
END_VAR
VAR
	pDatatypeAddedEvent : POINTER TO DatatypeAddedEvent;
END_VAR
pDatatypeAddedEvent := __NEW(DatatypeAddedEvent(Target := Datatype));
eventEmitter.Emit('OnDatatypeAdded',pDatatypeAddedEvent^);
pDatatypeAddedEvent^.Dispose();
END_METHOD

METHOD PROTECTED EmitOnEnumDatatypeAddedEvent
VAR_INPUT
	Datatype : I_EnumDatatype;
END_VAR
VAR
	pEnumDatatypeAddedEvent : POINTER TO EnumDatatypeAddedEvent;
END_VAR
pEnumDatatypeAddedEvent := __NEW(EnumDatatypeAddedEvent(Target := Datatype));
eventEmitter.Emit('OnDatatypeAdded',pEnumDatatypeAddedEvent^);
pEnumDatatypeAddedEvent^.Dispose();
END_METHOD

METHOD PROTECTED EmitOnStructuredDatatypeAddedEvent
VAR_INPUT
	Datatype : I_StructuredDatatype;
END_VAR
VAR
	pStructuredDatatypeAddedEvent : POINTER TO StructuredDatatypeAddedEvent;
END_VAR
pStructuredDatatypeAddedEvent := __NEW(StructuredDatatypeAddedEvent(Target := Datatype));
eventEmitter.Emit('OnDatatypeAdded',pStructuredDatatypeAddedEvent^);
pStructuredDatatypeAddedEvent^.Dispose();
END_METHOD

METHOD PUBLIC Accept
VAR_INPUT
	Visitor : I_DatatypeVisitor;
END_VAR
AcceptPrimative(Visitor);
AcceptStructures(Visitor);
AcceptAlias(Visitor);
AcceptEnum(Visitor);
END_METHOD

METHOD PUBLIC GetAliasByIdentifier : BOOL
VAR_INPUT
	Identifier : T_MAXSTRING;
	Destination : REFERENCE TO I_AliasDatatype;
END_VAR
GetAliasByIdentifier := alias.TryGetValue(Identifier, Destination);
END_METHOD

METHOD PUBLIC GetEnumByIdentifier : BOOL
VAR_INPUT
	Identifier : T_MAXSTRING;
	Destination : REFERENCE TO I_EnumDatatype;
END_VAR
GetEnumByIdentifier := enums.TryGetValue(Identifier, Destination);
END_METHOD

METHOD PUBLIC GetPrimitiveByTypeName : BOOL
VAR_INPUT
	TypeName : T_MAXSTRING;
	Destination : REFERENCE TO I_AliasDatatype;
END_VAR
GetPrimitiveByTypeName := primitives.TryGetValue(TypeName, Destination);
END_METHOD

METHOD PUBLIC GetStructureByIdentifier : BOOL
VAR_INPUT
	Identifier : T_MAXSTRING;
	Destination : REFERENCE TO I_StructuredDatatype;
END_VAR
GetStructureByIdentifier := structures.TryGetValue(Identifier, Destination);
END_METHOD

METHOD PUBLIC OffEvent
VAR_INPUT
	EventName : T_MaxString;
	EventHandler : I_EventHandler;
END_VAR
eventEmitter.OffEvent(EventName, EventHandler);
END_METHOD

METHOD PUBLIC OnceEvent
VAR_INPUT
	EventName : T_MaxString;
	EventHandler : I_EventHandler;
END_VAR
eventEmitter.OnceEvent(EventName, EventHandler);
END_METHOD

METHOD PUBLIC OnEvent
VAR_INPUT
	EventName : T_MaxString;
	EventHandler : I_EventHandler;
END_VAR
eventEmitter.OnEvent(EventName, EventHandler);
END_METHOD

METHOD RegisterDatatype
VAR_INPUT
	Datatype : I_Datatype;
END_VAR
VAR
	datatypeAsStructure : I_StructuredDatatype;
	datatypeAsAlias : I_AliasDatatype;
	datatypeAsEnum : I_EnumDatatype;
END_VAR
IF Datatype.TryResolveAsStructuredDatatype(datatypeAsStructure) THEN
	structures.AddOrUpdate(datatypeAsStructure.Identifier, datatypeAsStructure);
	emitOnStructuredDatatypeAddedEvent(datatypeAsStructure);
	RETURN;
END_IF

IF Datatype.TryResolveAsAliasDatatype(datatypeAsAlias) THEN
	alias.AddOrUpdate(datatypeAsAlias.Identifier, datatypeAsAlias);
	emitOnAliasDatatypeAddedEvent(datatypeAsAlias);
	RETURN;
END_IF

IF Datatype.TryResolveAsEnumDatatype(datatypeAsEnum) THEN
	enums.AddOrUpdate(datatypeAsEnum.Identifier, datatypeAsEnum);
	emitOnEnumDatatypeAddedEvent(datatypeAsEnum);
	RETURN;
END_IF

// add arrays

primitives.AddOrUpdate(Datatype.TypeName, Datatype);
emitOnDatatypeAddedEvent(Datatype);
END_METHOD

METHOD PUBLIC SerializeTypeWith
VAR_INPUT
	Serializer : I_Serializer;
END_VAR
Serializer.StartObject();
Serializer.AddKey('datatypes');
Serializer.StartArray();
SerializePrimitiveTypeWith(Serializer);
SerializeStructuresTypeWith(Serializer);
SerializeAliasTypeWith(Serializer);
SerializeEnumsTypeWith(Serializer);
Serializer.EndArray();
Serializer.EndObject();
END_METHOD

END_FUNCTION_BLOCK

// Datatypes/Interface/I_Datatypes
INTERFACE I_Datatypes EXTENDS I_EventEmitter

METHOD PUBLIC Accept
VAR_INPUT
	Visitor : I_DatatypeVisitor;
END_VAR
END_METHOD

METHOD PUBLIC GetAliasByIdentifier : BOOL
VAR_INPUT
	Identifier : T_MAXSTRING;
	Destination : REFERENCE TO I_AliasDatatype;
END_VAR
END_METHOD

METHOD PUBLIC GetPrimitiveByTypeName : BOOL
VAR_INPUT
	TypeName : T_MAXSTRING;
	Destination : REFERENCE TO I_AliasDatatype;
END_VAR
END_METHOD

METHOD PUBLIC GetStructureByIdentifier : BOOL
VAR_INPUT
	Identifier : T_MAXSTRING;
	Destination : REFERENCE TO I_StructuredDatatype;
END_VAR
END_METHOD

METHOD RegisterDatatype
VAR_INPUT
	Datatype : I_Datatype;
END_VAR
END_METHOD

METHOD PUBLIC SerializeTypeWith
VAR_INPUT
	Serializer : I_Serializer;
END_VAR
END_METHOD

END_INTERFACE

// Primitive/_BOOL
{attribute 'linkalways'} 
{attribute 'no_explicit_call' := 'This FB is a CLASS and must be accessed using methods or properties'}
{attribute 'enable_dynamic_creation'}
FUNCTION_BLOCK _BOOL EXTENDS DatatypeBase
VAR
	localData : BOOL;
	activeData : REFERENCE TO BOOL REF= localData;
END_VAR

METHOD FB_init : BOOL
VAR_INPUT
	bInitRetains : BOOL; // if TRUE, the retain variables are initialized (warm start / cold start)
	bInCopyCode : BOOL;  // if TRUE, the instance afterwards gets moved into the copy code (online change)
	InitialValue : BOOL;
END_VAR
localData := InitialValue;
END_METHOD

PROPERTY PUBLIC Address : PVOID
GET
Address := ADR(activeData);
END_GET
END_PROPERTY

METHOD PUBLIC ClearReference
VAR_INPUT
END_VAR
activeData REF= localData;
END_METHOD

METHOD PUBLIC Clone : I_Datatype
VAR
    pClone : POINTER TO _BOOL;
END_VAR
pClone := __NEW(_BOOL(InitialValue := Value));
Clone := pClone^;
END_METHOD

METHOD PUBLIC MakeReferenceTo
VAR_INPUT
	ReferenceTarget : REFERENCE TO BOOL;
END_VAR
activeData REF= ReferenceTarget;
END_METHOD

METHOD PUBLIC SerializeWith
VAR_INPUT
	Serializer : I_Serializer;
END_VAR
Serializer.AddBool(activeData);
END_METHOD

PROPERTY PUBLIC Size : UDINT
GET
Size := SIZEOF(activeData);
END_GET
END_PROPERTY

METHOD TryDeserializeFrom : BOOL
VAR_INPUT
	Deserializer : I_Deserializer;
	Feedback : I_DeserializerFeedback;
END_VAR
TryDeserializeFrom := Deserializer.TryGetBool(activeData, Feedback);
END_METHOD

METHOD TryMakeReferenceTo : BOOL
VAR_INPUT
	Target : I_Datatype;
END_VAR
VAR
	pTargetData : POINTER TO BOOL;
END_VAR
IF NOT (Target.TypeName = TypeName) THEN
	RETURN;
END_IF

pTargetData := Target.Address;
activeData REF= pTargetData^;
TryMakeReferenceTo := TRUE;
END_METHOD

PROPERTY PUBLIC TypeName : T_MAXSTRING
GET
TypeName := 'BOOL';
END_GET
END_PROPERTY

PROPERTY PUBLIC Value : BOOL
GET
Value := activeData;
END_GET
SET
activeData := Value;
END_SET
END_PROPERTY

END_FUNCTION_BLOCK

// Primitive/_BYTE
{attribute 'linkalways'} 
{attribute 'no_explicit_call' := 'This FB is a CLASS and must be accessed using methods or properties'}
{attribute 'enable_dynamic_creation'}
FUNCTION_BLOCK _BYTE EXTENDS NumericDatatypeBase
VAR
	localData : BYTE;
	activeData : REFERENCE TO BYTE REF= localData;
END_VAR

METHOD FB_init : BOOL
VAR_INPUT
	bInitRetains : BOOL; // if TRUE, the retain variables are initialized (warm start / cold start)
	bInCopyCode : BOOL;  // if TRUE, the instance afterwards gets moved into the copy code (online change)
	InitialValue : BYTE;
END_VAR
localData := InitialValue;
END_METHOD

METHOD PROTECTED SerializeMaxValue
VAR_INPUT
	Serializer : I_Serializer;
END_VAR
Serializer.AddByte(MaxValue);
END_METHOD

METHOD PROTECTED SerializeMinValue
VAR_INPUT
	Serializer : I_Serializer;
END_VAR
Serializer.AddByte(MinValue);
END_METHOD

PROPERTY PUBLIC Address : PVOID
GET
Address := ADR(activeData);
END_GET
END_PROPERTY

METHOD PUBLIC ClearReference
VAR_INPUT
END_VAR
activeData REF= localData;
END_METHOD

METHOD PUBLIC Clone : I_Datatype
VAR
    pClone : POINTER TO _BYTE;
END_VAR
pClone := __NEW(_BYTE(InitialValue := Value));
Clone := pClone^;
END_METHOD

PROPERTY PUBLIC IsFloat : BOOL
GET
IsFloat := FALSE;
END_GET
END_PROPERTY

PROPERTY PUBLIC IsSigned : BOOL
GET
IsSigned := FALSE;
END_GET
END_PROPERTY

METHOD PUBLIC MakeReferenceTo
VAR_INPUT
	ReferenceTarget : REFERENCE TO BYTE;
END_VAR
activeData REF= ReferenceTarget;
END_METHOD

PROPERTY PUBLIC MaxValue : BYTE
GET
MaxValue := DatatypeLimits.BYTE_MAX_VALUE;
END_GET
END_PROPERTY

PROPERTY PUBLIC MinValue : BYTE
GET
MinValue := DatatypeLimits.BYTE_MIN_VALUE;
END_GET
END_PROPERTY

METHOD PUBLIC SerializeWith
VAR_INPUT
	Serializer : I_Serializer;
END_VAR
Serializer.AddByte(activeData);
END_METHOD

PROPERTY PUBLIC Size : UDINT
GET
Size := SIZEOF(activeData);
END_GET
END_PROPERTY

METHOD TryDeserializeFrom : BOOL
VAR_INPUT
	Deserializer : I_Deserializer;
	Feedback : I_DeserializerFeedback;
END_VAR
TryDeserializeFrom := Deserializer.TryGetByte(activeData, Feedback);
END_METHOD

METHOD TryMakeReferenceTo : BOOL
VAR_INPUT
	Target : I_Datatype;
END_VAR
VAR
	pTargetData : POINTER TO BYTE;
END_VAR
IF NOT (Target.TypeName = TypeName) THEN
	RETURN;
END_IF

pTargetData := Target.Address;
activeData REF= pTargetData^;
TryMakeReferenceTo := TRUE;
END_METHOD

PROPERTY PUBLIC TypeName : T_MAXSTRING
GET
TypeName := 'BYTE';
END_GET
END_PROPERTY

PROPERTY PUBLIC Value : BYTE
GET
Value := activeData;
END_GET
SET
activeData := Value;
END_SET
END_PROPERTY

END_FUNCTION_BLOCK

// Primitive/_DINT
{attribute 'linkalways'} 
{attribute 'no_explicit_call' := 'This FB is a CLASS and must be accessed using methods or properties'}
{attribute 'enable_dynamic_creation'}
FUNCTION_BLOCK _DINT EXTENDS NumericDatatypeBase
VAR
	localData : DINT;
	activeData : REFERENCE TO DINT REF= localData;
END_VAR

METHOD FB_init : BOOL
VAR_INPUT
	bInitRetains : BOOL; // if TRUE, the retain variables are initialized (warm start / cold start)
	bInCopyCode : BOOL;  // if TRUE, the instance afterwards gets moved into the copy code (online change)
	InitialValue : DINT;
END_VAR
localData := InitialValue;
END_METHOD

METHOD PROTECTED SerializeMaxValue
VAR_INPUT
	Serializer : I_Serializer;
END_VAR
Serializer.AddDint(MaxValue);
END_METHOD

METHOD PROTECTED SerializeMinValue
VAR_INPUT
	Serializer : I_Serializer;
END_VAR
Serializer.AddDint(MinValue);
END_METHOD

PROPERTY PUBLIC Address : PVOID
GET
Address := ADR(activeData);
END_GET
END_PROPERTY

METHOD PUBLIC ClearReference
VAR_INPUT
END_VAR
activeData REF= localData;
END_METHOD

METHOD PUBLIC Clone : I_Datatype
VAR
    pClone : POINTER TO _DINT;
END_VAR
pClone := __NEW(_DINT(InitialValue := Value));
Clone := pClone^;
END_METHOD

PROPERTY PUBLIC IsFloat : BOOL
GET
IsFloat := FALSE;
END_GET
END_PROPERTY

PROPERTY PUBLIC IsSigned : BOOL
GET
IsSigned := TRUE;
END_GET
END_PROPERTY

METHOD PUBLIC MakeReferenceTo
VAR_INPUT
	ReferenceTarget : REFERENCE TO DINT;
END_VAR
activeData REF= ReferenceTarget;
END_METHOD

PROPERTY PUBLIC MaxValue : DINT
GET
MaxValue := DatatypeLimits.DINT_MAX_VALUE;
END_GET
END_PROPERTY

PROPERTY PUBLIC MinValue : DINT
GET
MinValue := DatatypeLimits.DINT_MIN_VALUE;
END_GET
END_PROPERTY

METHOD PUBLIC SerializeWith
VAR_INPUT
	Serializer : I_Serializer;
END_VAR
Serializer.AddDint(activeData);
END_METHOD

PROPERTY PUBLIC Size : UDINT
GET
Size := SIZEOF(activeData);
END_GET
END_PROPERTY

METHOD TryDeserializeFrom : BOOL
VAR_INPUT
	Deserializer : I_Deserializer;
	Feedback : I_DeserializerFeedback;
END_VAR
TryDeserializeFrom := Deserializer.TryGetDint(activeData, Feedback);
END_METHOD

METHOD TryMakeReferenceTo : BOOL
VAR_INPUT
	Target : I_Datatype;
END_VAR
VAR
	pTargetData : POINTER TO DINT;
END_VAR
IF NOT (Target.TypeName = TypeName) THEN
	RETURN;
END_IF

pTargetData := Target.Address;
activeData REF= pTargetData^;
TryMakeReferenceTo := TRUE;
END_METHOD

PROPERTY PUBLIC TypeName : T_MAXSTRING
GET
TypeName := 'DINT';
END_GET
END_PROPERTY

PROPERTY PUBLIC Value : DINT
GET
Value := activeData;
END_GET
SET
activeData := Value;
END_SET
END_PROPERTY

END_FUNCTION_BLOCK

// Primitive/_DT
{attribute 'linkalways'} 
{attribute 'no_explicit_call' := 'This FB is a CLASS and must be accessed using methods or properties'}
{attribute 'enable_dynamic_creation'}
FUNCTION_BLOCK _DT EXTENDS DatatypeBase
VAR
	localData : DT;
	activeData : REFERENCE TO DT REF= localData;
END_VAR

METHOD FB_init : BOOL
VAR_INPUT
	bInitRetains : BOOL; // if TRUE, the retain variables are initialized (warm start / cold start)
	bInCopyCode : BOOL;  // if TRUE, the instance afterwards gets moved WORDo the copy code (online change)
	InitialValue : DT;
END_VAR
localData := InitialValue;
END_METHOD

PROPERTY PUBLIC Address : PVOID
GET
Address := ADR(activeData);
END_GET
END_PROPERTY

METHOD PUBLIC ClearReference
VAR_INPUT
END_VAR
activeData REF= localData;
END_METHOD

METHOD PUBLIC Clone : I_Datatype
VAR
    pClone : POINTER TO _DT;
END_VAR
pClone := __NEW(_DT(InitialValue := Value));
Clone := pClone^;
END_METHOD

METHOD PUBLIC MakeReferenceTo
VAR_INPUT
	ReferenceTarget : REFERENCE TO DT;
END_VAR
activeData REF= ReferenceTarget;
END_METHOD

METHOD PUBLIC SerializeWith
VAR_INPUT
	Serializer : I_Serializer;
END_VAR
Serializer.AddDateTime(activeData);
END_METHOD

PROPERTY PUBLIC Size : UDINT
GET
Size := SIZEOF(activeData);
END_GET
END_PROPERTY

METHOD TryDeserializeFrom : BOOL
VAR_INPUT
	Deserializer : I_Deserializer;
	Feedback : I_DeserializerFeedback;
END_VAR
TryDeserializeFrom := Deserializer.TryGetDateTime(activeData, Feedback);
END_METHOD

METHOD TryMakeReferenceTo : BOOL
VAR_INPUT
	Target : I_Datatype;
END_VAR
VAR
	pTargetData : POINTER TO DT;
END_VAR
IF NOT (Target.TypeName = TypeName) THEN
	RETURN;
END_IF

pTargetData := Target.Address;
activeData REF= pTargetData^;
TryMakeReferenceTo := TRUE;
END_METHOD

PROPERTY PUBLIC TypeName : T_MAXSTRING
GET
TypeName := 'DT';
END_GET
END_PROPERTY

PROPERTY PUBLIC Value : DT
GET
Value := activeData;
END_GET
SET
activeData := Value;
END_SET
END_PROPERTY

END_FUNCTION_BLOCK

// Primitive/_DWORD
{attribute 'linkalways'} 
{attribute 'no_explicit_call' := 'This FB is a CLASS and must be accessed using methods or properties'}
{attribute 'enable_dynamic_creation'}
FUNCTION_BLOCK _DWORD EXTENDS NumericDatatypeBase
VAR
	localData : DWORD;
	activeData : REFERENCE TO DWORD REF= localData;
END_VAR

METHOD FB_init : BOOL
VAR_INPUT
	bInitRetains : BOOL; // if TRUE, the retain variables are initialized (warm start / cold start)
	bInCopyCode : BOOL;  // if TRUE, the instance afterwards gets moved WORDo the copy code (online change)
	InitialValue : DWORD;
END_VAR
localData := InitialValue;
END_METHOD

METHOD PROTECTED SerializeMaxValue
VAR_INPUT
	Serializer : I_Serializer;
END_VAR
Serializer.AddDword(MaxValue);
END_METHOD

METHOD PROTECTED SerializeMinValue
VAR_INPUT
	Serializer : I_Serializer;
END_VAR
Serializer.AddDword(MinValue);
END_METHOD

PROPERTY PUBLIC Address : PVOID
GET
Address := ADR(activeData);
END_GET
END_PROPERTY

METHOD PUBLIC ClearReference
VAR_INPUT
END_VAR
activeData REF= localData;
END_METHOD

METHOD PUBLIC Clone : I_Datatype
VAR
    pClone : POINTER TO _DWORD;
END_VAR
pClone := __NEW(_DWORD(InitialValue := Value));
Clone := pClone^;
END_METHOD

PROPERTY PUBLIC IsFloat : BOOL
GET
IsFloat := FALSE;
END_GET
END_PROPERTY

PROPERTY PUBLIC IsSigned : BOOL
GET
IsSigned := FALSE;
END_GET
END_PROPERTY

METHOD PUBLIC MakeReferenceTo
VAR_INPUT
	ReferenceTarget : REFERENCE TO DWORD;
END_VAR
activeData REF= ReferenceTarget;
END_METHOD

PROPERTY PUBLIC MaxValue : DWORD
GET
MaxValue := DatatypeLimits.DWORD_MAX_VALUE;
END_GET
END_PROPERTY

PROPERTY PUBLIC MinValue : DWORD
GET
MinValue := DatatypeLimits.DWORD_MIN_VALUE;
END_GET
END_PROPERTY

METHOD PUBLIC SerializeWith
VAR_INPUT
	Serializer : I_Serializer;
END_VAR
Serializer.AddDword(activeData);
END_METHOD

PROPERTY PUBLIC Size : UDINT
GET
Size := SIZEOF(activeData);
END_GET
END_PROPERTY

METHOD TryDeserializeFrom : BOOL
VAR_INPUT
	Deserializer : I_Deserializer;
	Feedback : I_DeserializerFeedback;
END_VAR
TryDeserializeFrom := Deserializer.TryGetDword(activeData, Feedback);
END_METHOD

METHOD TryMakeReferenceTo : BOOL
VAR_INPUT
	Target : I_Datatype;
END_VAR
VAR
	pTargetData : POINTER TO DWORD;
END_VAR
IF NOT (Target.TypeName = TypeName) THEN
	RETURN;
END_IF

pTargetData := Target.Address;
activeData REF= pTargetData^;
TryMakeReferenceTo := TRUE;
END_METHOD

PROPERTY PUBLIC TypeName : T_MAXSTRING
GET
TypeName := 'DWORD';
END_GET
END_PROPERTY

PROPERTY PUBLIC Value : DWORD
GET
Value := activeData;
END_GET
SET
activeData := Value;
END_SET
END_PROPERTY

END_FUNCTION_BLOCK

// Primitive/_INT
{attribute 'linkalways'} 
{attribute 'no_explicit_call' := 'This FB is a CLASS and must be accessed using methods or properties'}
{attribute 'enable_dynamic_creation'}
FUNCTION_BLOCK _INT EXTENDS NumericDatatypeBase
VAR
	localData : INT;
	activeData : REFERENCE TO INT REF= localData;
END_VAR

METHOD FB_init : BOOL
VAR_INPUT
	bInitRetains : BOOL; // if TRUE, the retain variables are initialized (warm start / cold start)
	bInCopyCode : BOOL;  // if TRUE, the instance afterwards gets moved into the copy code (online change)
	InitialValue : INT;
END_VAR
localData := InitialValue;
END_METHOD

METHOD PROTECTED SerializeMaxValue
VAR_INPUT
	Serializer : I_Serializer;
END_VAR
Serializer.AddInt(MaxValue);
END_METHOD

METHOD PROTECTED SerializeMinValue
VAR_INPUT
	Serializer : I_Serializer;
END_VAR
Serializer.AddInt(MinValue);
END_METHOD

PROPERTY PUBLIC Address : PVOID
GET
Address := ADR(activeData);
END_GET
END_PROPERTY

METHOD PUBLIC ClearReference
VAR_INPUT
END_VAR
activeData REF= localData;
END_METHOD

METHOD PUBLIC Clone : I_Datatype
VAR
    pClone : POINTER TO _INT;
END_VAR
pClone := __NEW(_INT(InitialValue := Value));
Clone := pClone^;
END_METHOD

PROPERTY PUBLIC IsFloat : BOOL
GET
IsFloat := FALSE;
END_GET
END_PROPERTY

PROPERTY PUBLIC IsSigned : BOOL
GET
IsSigned := TRUE;
END_GET
END_PROPERTY

METHOD PUBLIC MakeReferenceTo
VAR_INPUT
	ReferenceTarget : REFERENCE TO INT;
END_VAR
activeData REF= ReferenceTarget;
END_METHOD

PROPERTY PUBLIC MaxValue : INT
GET
MaxValue := DatatypeLimits.INT_MAX_VALUE;
END_GET
END_PROPERTY

PROPERTY PUBLIC MinValue : INT
GET
MinValue := DatatypeLimits.INT_MIN_VALUE;
END_GET
END_PROPERTY

METHOD PUBLIC SerializeWith
VAR_INPUT
	Serializer : I_Serializer;
END_VAR
Serializer.AddInt(activeData);
END_METHOD

PROPERTY PUBLIC Size : UDINT
GET
Size := SIZEOF(activeData);
END_GET
END_PROPERTY

METHOD TryDeserializeFrom : BOOL
VAR_INPUT
	Deserializer : I_Deserializer;
	Feedback : I_DeserializerFeedback;
END_VAR
TryDeserializeFrom := Deserializer.TryGetInt(activeData, Feedback);
END_METHOD

METHOD TryMakeReferenceTo : BOOL
VAR_INPUT
	Target : I_Datatype;
END_VAR
VAR
	pTargetData : POINTER TO INT;
END_VAR
IF NOT (Target.TypeName = TypeName) THEN
	RETURN;
END_IF

pTargetData := Target.Address;
activeData REF= pTargetData^;
TryMakeReferenceTo := TRUE;
END_METHOD

PROPERTY PUBLIC TypeName : T_MAXSTRING
GET
TypeName := 'INT';
END_GET
END_PROPERTY

PROPERTY PUBLIC Value : INT
GET
Value := activeData;
END_GET
SET
activeData := Value;
END_SET
END_PROPERTY

END_FUNCTION_BLOCK

// Primitive/_LINT
{attribute 'linkalways'} 
{attribute 'no_explicit_call' := 'This FB is a CLASS and must be accessed using methods or properties'}
{attribute 'enable_dynamic_creation'}
FUNCTION_BLOCK _LINT EXTENDS NumericDatatypeBase
VAR
	localData : LINT;
	activeData : REFERENCE TO LINT REF= localData;
END_VAR

METHOD FB_init : BOOL
VAR_INPUT
	bInitRetains : BOOL; // if TRUE, the retain variables are initialized (warm start / cold start)
	bInCopyCode : BOOL;  // if TRUE, the instance afterwards gets moved into the copy code (online change)
	InitialValue : LINT;
END_VAR
localData := InitialValue;
END_METHOD

METHOD PROTECTED SerializeMaxValue
VAR_INPUT
	Serializer : I_Serializer;
END_VAR
Serializer.AddLint(MaxValue);
END_METHOD

METHOD PROTECTED SerializeMinValue
VAR_INPUT
	Serializer : I_Serializer;
END_VAR
Serializer.AddLint(MinValue);
END_METHOD

PROPERTY PUBLIC Address : PVOID
GET
Address := ADR(activeData);
END_GET
END_PROPERTY

METHOD PUBLIC ClearReference
VAR_INPUT
END_VAR
activeData REF= localData;
END_METHOD

METHOD PUBLIC Clone : I_Datatype
VAR
    pClone : POINTER TO _LINT;
END_VAR
pClone := __NEW(_LINT(InitialValue := Value));
Clone := pClone^;
END_METHOD

PROPERTY PUBLIC IsFloat : BOOL
GET
IsFloat := FALSE;
END_GET
END_PROPERTY

PROPERTY PUBLIC IsSigned : BOOL
GET
IsSigned := TRUE;
END_GET
END_PROPERTY

METHOD PUBLIC MakeReferenceTo
VAR_INPUT
	ReferenceTarget : REFERENCE TO LINT;
END_VAR
activeData REF= ReferenceTarget;
END_METHOD

PROPERTY PUBLIC MaxValue : LINT
GET
MaxValue :=  DatatypeLimits.LINT_MAX_VALUE;
END_GET
END_PROPERTY

PROPERTY PUBLIC MinValue : LINT
GET
MinValue := DatatypeLimits.LINT_MIN_VALUE;
END_GET
END_PROPERTY

METHOD PUBLIC SerializeWith
VAR_INPUT
	Serializer : I_Serializer;
END_VAR
Serializer.AddLint(activeData);
END_METHOD

PROPERTY PUBLIC Size : UDINT
GET
Size := SIZEOF(activeData);
END_GET
END_PROPERTY

METHOD TryDeserializeFrom : BOOL
VAR_INPUT
	Deserializer : I_Deserializer;
	Feedback : I_DeserializerFeedback;
END_VAR
TryDeserializeFrom := Deserializer.TryGetLint(activeData, Feedback);
END_METHOD

METHOD TryMakeReferenceTo : BOOL
VAR_INPUT
	Target : I_Datatype;
END_VAR
VAR
	pTargetData : POINTER TO LINT;
END_VAR
IF NOT (Target.TypeName = TypeName) THEN
	RETURN;
END_IF

pTargetData := Target.Address;
activeData REF= pTargetData^;
TryMakeReferenceTo := TRUE;
END_METHOD

PROPERTY PUBLIC TypeName : T_MAXSTRING
GET
TypeName := 'LINT';
END_GET
END_PROPERTY

PROPERTY PUBLIC Value : LINT
GET
Value := activeData;
END_GET
SET
activeData := Value;
END_SET
END_PROPERTY

END_FUNCTION_BLOCK

// Primitive/_LREAL
{attribute 'linkalways'} 
{attribute 'no_explicit_call' := 'This FB is a CLASS and must be accessed using methods or properties'}
{attribute 'enable_dynamic_creation'}
FUNCTION_BLOCK _LREAL EXTENDS NumericDatatypeBase
VAR
	localData : LREAL;
	activeData : REFERENCE TO LREAL REF= localData;
END_VAR

METHOD FB_init : BOOL
VAR_INPUT
	bInitRetains : BOOL; // if TRUE, the retain variables are initialized (warm start / cold start)
	bInCopyCode : BOOL;  // if TRUE, the instance afterwards gets moved into the copy code (online change)
	InitialValue : LREAL;
END_VAR
localData := InitialValue;
END_METHOD

METHOD PROTECTED SerializeMaxValue
VAR_INPUT
	Serializer : I_Serializer;
END_VAR
Serializer.AddLreal(MaxValue);
END_METHOD

METHOD PROTECTED SerializeMinValue
VAR_INPUT
	Serializer : I_Serializer;
END_VAR
Serializer.AddLreal(MinValue);
END_METHOD

PROPERTY PUBLIC Address : PVOID
GET
Address := ADR(activeData);
END_GET
END_PROPERTY

METHOD PUBLIC ClearReference
VAR_INPUT
END_VAR
activeData REF= localData;
END_METHOD

METHOD PUBLIC Clone : I_Datatype
VAR
    pClone : POINTER TO _LREAL;
END_VAR
pClone := __NEW(_LREAL(InitialValue := Value));
Clone := pClone^;
END_METHOD

PROPERTY PUBLIC IsFloat : BOOL
GET
IsFloat := TRUE;
END_GET
END_PROPERTY

PROPERTY PUBLIC IsSigned : BOOL
GET
IsSigned := TRUE;
END_GET
END_PROPERTY

METHOD PUBLIC MakeReferenceTo
VAR_INPUT
	ReferenceTarget : REFERENCE TO LREAL;
END_VAR
activeData REF= ReferenceTarget;
END_METHOD

PROPERTY PUBLIC MaxValue : LREAL
GET
MaxValue :=  DatatypeLimits.LREAL_MAX_VALUE;
END_GET
END_PROPERTY

PROPERTY PUBLIC MinValue : LREAL
GET
MinValue := DatatypeLimits.LREAL_MIN_VALUE;
END_GET
END_PROPERTY

METHOD PUBLIC SerializeWith
VAR_INPUT
	Serializer : I_Serializer;
END_VAR
Serializer.AddLreal(activeData);
END_METHOD

PROPERTY PUBLIC Size : UDINT
GET
Size := SIZEOF(activeData);
END_GET
END_PROPERTY

METHOD TryDeserializeFrom : BOOL
VAR_INPUT
	Deserializer : I_Deserializer;
	Feedback : I_DeserializerFeedback;
END_VAR
TryDeserializeFrom := Deserializer.TryGetLreal(activeData, Feedback);
END_METHOD

METHOD TryMakeReferenceTo : BOOL
VAR_INPUT
	Target : I_Datatype;
END_VAR
VAR
	pTargetData : POINTER TO LREAL;
END_VAR
IF NOT (Target.TypeName = TypeName) THEN
	RETURN;
END_IF

pTargetData := Target.Address;
activeData REF= pTargetData^;
TryMakeReferenceTo := TRUE;
END_METHOD

PROPERTY PUBLIC TypeName : T_MAXSTRING
GET
TypeName := 'LREAL';
END_GET
END_PROPERTY

PROPERTY PUBLIC Value : LREAL
GET
Value := activeData;
END_GET
SET
activeData := Value;
END_SET
END_PROPERTY

END_FUNCTION_BLOCK

// Primitive/_LWORD
{attribute 'linkalways'} 
{attribute 'no_explicit_call' := 'This FB is a CLASS and must be accessed using methods or properties'}
{attribute 'enable_dynamic_creation'}
FUNCTION_BLOCK _LWORD EXTENDS NumericDatatypeBase
VAR
	localData : LWORD;
	activeData : REFERENCE TO LWORD REF= localData;
END_VAR

METHOD FB_init : BOOL
VAR_INPUT
	bInitRetains : BOOL; // if TRUE, the retain variables are initialized (warm start / cold start)
	bInCopyCode : BOOL;  // if TRUE, the instance afterwards gets moved WORDo the copy code (online change)
	InitialValue : LWORD;
END_VAR
localData := InitialValue;
END_METHOD

METHOD PROTECTED SerializeMaxValue
VAR_INPUT
	Serializer : I_Serializer;
END_VAR
Serializer.AddLword(MaxValue);
END_METHOD

METHOD PROTECTED SerializeMinValue
VAR_INPUT
	Serializer : I_Serializer;
END_VAR
Serializer.AddLword(MinValue);
END_METHOD

PROPERTY PUBLIC Address : PVOID
GET
Address := ADR(activeData);
END_GET
END_PROPERTY

METHOD PUBLIC ClearReference
VAR_INPUT
END_VAR
activeData REF= localData;
END_METHOD

METHOD PUBLIC Clone : I_Datatype
VAR
    pClone : POINTER TO _LWORD;
END_VAR
pClone := __NEW(_LWORD(InitialValue := Value));
Clone := pClone^;
END_METHOD

PROPERTY PUBLIC IsFloat : BOOL
GET
IsFloat := FALSE;
END_GET
END_PROPERTY

PROPERTY PUBLIC IsSigned : BOOL
GET
IsSigned := FALSE;
END_GET
END_PROPERTY

METHOD PUBLIC MakeReferenceTo
VAR_INPUT
	ReferenceTarget : REFERENCE TO LWORD;
END_VAR
activeData REF= ReferenceTarget;
END_METHOD

PROPERTY PUBLIC MaxValue : LWORD
GET
MaxValue :=  DatatypeLimits.LWORD_MAX_VALUE;
END_GET
END_PROPERTY

PROPERTY PUBLIC MinValue : LWORD
GET
MinValue := DatatypeLimits.LWORD_MIN_VALUE;
END_GET
END_PROPERTY

METHOD PUBLIC SerializeWith
VAR_INPUT
	Serializer : I_Serializer;
END_VAR
Serializer.AddLword(activeData);
END_METHOD

PROPERTY PUBLIC Size : UDINT
GET
Size := SIZEOF(activeData);
END_GET
END_PROPERTY

METHOD TryDeserializeFrom : BOOL
VAR_INPUT
	Deserializer : I_Deserializer;
	Feedback : I_DeserializerFeedback;
END_VAR
TryDeserializeFrom := Deserializer.TryGetLword(activeData, Feedback);
END_METHOD

METHOD TryMakeReferenceTo : BOOL
VAR_INPUT
	Target : I_Datatype;
END_VAR
VAR
	pTargetData : POINTER TO LWORD;
END_VAR
IF NOT (Target.TypeName = TypeName) THEN
	RETURN;
END_IF

pTargetData := Target.Address;
activeData REF= pTargetData^;
TryMakeReferenceTo := TRUE;
END_METHOD

PROPERTY PUBLIC TypeName : T_MAXSTRING
GET
TypeName := 'LWORD';
END_GET
END_PROPERTY

PROPERTY PUBLIC Value : LWORD
GET
Value := activeData;
END_GET
SET
activeData := Value;
END_SET
END_PROPERTY

END_FUNCTION_BLOCK

// Primitive/_REAL
{attribute 'linkalways'} 
{attribute 'no_explicit_call' := 'This FB is a CLASS and must be accessed using methods or properties'}
{attribute 'enable_dynamic_creation'}
FUNCTION_BLOCK _REAL EXTENDS NumericDatatypeBase
VAR
	localData : REAL;
	activeData : REFERENCE TO REAL REF= localData;
END_VAR

METHOD FB_init : BOOL
VAR_INPUT
	bInitRetains : BOOL; // if TRUE, the retain variables are initialized (warm start / cold start)
	bInCopyCode : BOOL;  // if TRUE, the instance afterwards gets moved into the copy code (online change)
	InitialValue : REAL;
END_VAR
localData := InitialValue;
END_METHOD

METHOD PROTECTED SerializeMaxValue
VAR_INPUT
	Serializer : I_Serializer;
END_VAR
Serializer.AddReal(MaxValue);
END_METHOD

METHOD PROTECTED SerializeMinValue
VAR_INPUT
	Serializer : I_Serializer;
END_VAR
Serializer.AddReal(MinValue);
END_METHOD

PROPERTY PUBLIC Address : PVOID
GET
Address := ADR(activeData);
END_GET
END_PROPERTY

METHOD PUBLIC ClearReference
VAR_INPUT
END_VAR
activeData REF= localData;
END_METHOD

METHOD PUBLIC Clone : I_Datatype
VAR
    pClone : POINTER TO _REAL;
END_VAR
pClone := __NEW(_REAL(InitialValue := Value));
Clone := pClone^;
END_METHOD

PROPERTY PUBLIC IsFloat : BOOL
GET
IsFloat := TRUE;
END_GET
END_PROPERTY

PROPERTY PUBLIC IsSigned : BOOL
GET
IsSigned := TRUE;
END_GET
END_PROPERTY

METHOD PUBLIC MakeReferenceTo
VAR_INPUT
	ReferenceTarget : REFERENCE TO REAL;
END_VAR
activeData REF= ReferenceTarget;
END_METHOD

PROPERTY PUBLIC MaxValue : REAL
GET
MaxValue :=  DatatypeLimits.REAL_MAX_VALUE;
END_GET
END_PROPERTY

PROPERTY PUBLIC MinValue : REAL
GET
MinValue := DatatypeLimits.REAL_MIN_VALUE;
END_GET
END_PROPERTY

METHOD PUBLIC SerializeWith
VAR_INPUT
	Serializer : I_Serializer;
END_VAR
Serializer.AddReal(activeData);
END_METHOD

PROPERTY PUBLIC Size : UDINT
GET
Size := SIZEOF(activeData);
END_GET
END_PROPERTY

METHOD TryDeserializeFrom : BOOL
VAR_INPUT
	Deserializer : I_Deserializer;
	Feedback : I_DeserializerFeedback;
END_VAR
TryDeserializeFrom := Deserializer.TryGetReal(activeData, Feedback);
END_METHOD

METHOD TryMakeReferenceTo : BOOL
VAR_INPUT
	Target : I_Datatype;
END_VAR
VAR
	pTargetData : POINTER TO REAL;
END_VAR
IF NOT (Target.TypeName = TypeName) THEN
	RETURN;
END_IF

pTargetData := Target.Address;
activeData REF= pTargetData^;
TryMakeReferenceTo := TRUE;
END_METHOD

PROPERTY PUBLIC TypeName : T_MAXSTRING
GET
TypeName := 'REAL';
END_GET
END_PROPERTY

PROPERTY PUBLIC Value : REAL
GET
Value := activeData;
END_GET
SET
activeData := Value;
END_SET
END_PROPERTY

END_FUNCTION_BLOCK

// Primitive/_SINT
{attribute 'linkalways'} 
{attribute 'no_explicit_call' := 'This FB is a CLASS and must be accessed using methods or properties'}
{attribute 'enable_dynamic_creation'}
FUNCTION_BLOCK _SINT EXTENDS NumericDatatypeBase
VAR
	localData : SINT;
	activeData : REFERENCE TO SINT REF= localData;
END_VAR

METHOD FB_init : BOOL
VAR_INPUT
	bInitRetains : BOOL; // if TRUE, the retain variables are initialized (warm start / cold start)
	bInCopyCode : BOOL;  // if TRUE, the instance afterwards gets moved into the copy code (online change)
	InitialValue : SINT;
END_VAR
localData := InitialValue;
END_METHOD

METHOD PROTECTED SerializeMaxValue
VAR_INPUT
	Serializer : I_Serializer;
END_VAR
Serializer.AddSint(MaxValue);
END_METHOD

METHOD PROTECTED SerializeMinValue
VAR_INPUT
	Serializer : I_Serializer;
END_VAR
Serializer.AddSint(MinValue);
END_METHOD

PROPERTY PUBLIC Address : PVOID
GET
Address := ADR(activeData);
END_GET
END_PROPERTY

METHOD PUBLIC ClearReference
VAR_INPUT
END_VAR
activeData REF= localData;
END_METHOD

METHOD PUBLIC Clone : I_Datatype
VAR
    pClone : POINTER TO _SINT;
END_VAR
pClone := __NEW(_SINT(InitialValue := Value));
Clone := pClone^;
END_METHOD

PROPERTY PUBLIC IsFloat : BOOL
GET
IsFloat := FALSE;
END_GET
END_PROPERTY

PROPERTY PUBLIC IsSigned : BOOL
GET
IsSigned := TRUE;
END_GET
END_PROPERTY

METHOD PUBLIC MakeReferenceTo
VAR_INPUT
	ReferenceTarget : REFERENCE TO SINT;
END_VAR
activeData REF= ReferenceTarget;
END_METHOD

PROPERTY PUBLIC MaxValue : SINT
GET
MaxValue :=  DatatypeLimits.SINT_MAX_VALUE;
END_GET
END_PROPERTY

PROPERTY PUBLIC MinValue : SINT
GET
MinValue := DatatypeLimits.SINT_MIN_VALUE;
END_GET
END_PROPERTY

METHOD PUBLIC SerializeWith
VAR_INPUT
	Serializer : I_Serializer;
END_VAR
Serializer.AddSint(activeData);
END_METHOD

PROPERTY PUBLIC Size : UDINT
GET
Size := SIZEOF(activeData);
END_GET
END_PROPERTY

METHOD TryDeserializeFrom : BOOL
VAR_INPUT
	Deserializer : I_Deserializer;
	Feedback : I_DeserializerFeedback;
END_VAR
TryDeserializeFrom := Deserializer.TryGetSint(activeData, Feedback);
END_METHOD

METHOD TryMakeReferenceTo : BOOL
VAR_INPUT
	Target : I_Datatype;
END_VAR
VAR
	pTargetData : POINTER TO SINT;
END_VAR
IF NOT (Target.TypeName = TypeName) THEN
	RETURN;
END_IF

pTargetData := Target.Address;
activeData REF= pTargetData^;
TryMakeReferenceTo := TRUE;
END_METHOD

PROPERTY PUBLIC TypeName : T_MAXSTRING
GET
TypeName := 'SINT';
END_GET
END_PROPERTY

PROPERTY PUBLIC Value : SINT
GET
Value := activeData;
END_GET
SET
activeData := Value;
END_SET
END_PROPERTY

END_FUNCTION_BLOCK

// Primitive/_STRING
{attribute 'linkalways'} 
{attribute 'no_explicit_call' := 'This FB is a CLASS and must be accessed using methods or properties'}
{attribute 'enable_dynamic_creation'}
FUNCTION_BLOCK _STRING EXTENDS DatatypeBase
VAR
	localData : T_MaxString;
	activeData : REFERENCE TO T_MaxString REF= localData;
END_VAR

METHOD FB_init : BOOL
VAR_INPUT
	bInitRetains : BOOL; // if TRUE, the retain variables are initialized (warm start / cold start)
	bInCopyCode : BOOL;  // if TRUE, the instance afterwards gets moved WORDo the copy code (online change)
	InitialValue : T_MaxString;
END_VAR
localData := InitialValue;
END_METHOD

PROPERTY PUBLIC Address : PVOID
GET
Address := ADR(activeData);
END_GET
END_PROPERTY

METHOD PUBLIC ClearReference
VAR_INPUT
END_VAR
activeData REF= localData;
END_METHOD

METHOD PUBLIC Clone : I_Datatype
VAR
    pClone : POINTER TO _STRING;
END_VAR
pClone := __NEW(_STRING(InitialValue := Value));
Clone := pClone^;
END_METHOD

METHOD PUBLIC MakeReferenceTo
VAR_INPUT
	ReferenceTarget : REFERENCE TO T_MaxString;
END_VAR
activeData REF= ReferenceTarget;
END_METHOD

METHOD PUBLIC SerializeWith
VAR_INPUT
	Serializer : I_Serializer;
END_VAR
Serializer.AddString(activeData);
END_METHOD

PROPERTY PUBLIC Size : UDINT
GET
Size := SIZEOF(activeData);
END_GET
END_PROPERTY

METHOD TryDeserializeFrom : BOOL
VAR_INPUT
	Deserializer : I_Deserializer;
	Feedback : I_DeserializerFeedback;
END_VAR
TryDeserializeFrom := Deserializer.TryGetString(activeData, Feedback);
END_METHOD

METHOD TryMakeReferenceTo : BOOL
VAR_INPUT
	Target : I_Datatype;
END_VAR
VAR
	pTargetData : POINTER TO T_MaxString;
END_VAR
IF NOT (Target.TypeName = TypeName) THEN
	RETURN;
END_IF

pTargetData := Target.Address;
activeData REF= pTargetData^;
TryMakeReferenceTo := TRUE;
END_METHOD

PROPERTY PUBLIC TypeName : T_MAXSTRING
GET
TypeName := 'STRING';
END_GET
END_PROPERTY

PROPERTY PUBLIC Value : T_MaxString
GET
Value := activeData;
END_GET
SET
activeData := Value;
END_SET
END_PROPERTY

END_FUNCTION_BLOCK

// Primitive/_TIME_OF_DAY
{attribute 'linkalways'} 
{attribute 'no_explicit_call' := 'This FB is a CLASS and must be accessed using methods or properties'}
{attribute 'enable_dynamic_creation'}
FUNCTION_BLOCK _TIME_OF_DAY EXTENDS DatatypeBase
VAR
	localData : TIME_OF_DAY;
	activeData : REFERENCE TO TIME_OF_DAY REF= localData;
END_VAR

METHOD FB_init : BOOL
VAR_INPUT
	bInitRetains : BOOL; // if TRUE, the retain variables are initialized (warm start / cold start)
	bInCopyCode : BOOL;  // if TRUE, the instance afterwards gets moved WORDo the copy code (online change)
	InitialValue : TIME_OF_DAY;
END_VAR
localData := InitialValue;
END_METHOD

PROPERTY PUBLIC Address : PVOID
GET
Address := ADR(activeData);
END_GET
END_PROPERTY

METHOD PUBLIC ClearReference
VAR_INPUT
END_VAR
activeData REF= localData;
END_METHOD

METHOD PUBLIC Clone : I_Datatype
VAR
    pClone : POINTER TO _TIME_OF_DAY;
END_VAR
pClone := __NEW(_TIME_OF_DAY(InitialValue := Value));
Clone := pClone^;
END_METHOD

METHOD PUBLIC MakeReferenceTo
VAR_INPUT
	ReferenceTarget : REFERENCE TO TIME_OF_DAY;
END_VAR
activeData REF= ReferenceTarget;
END_METHOD

METHOD PUBLIC SerializeWith
VAR_INPUT
	Serializer : I_Serializer;
END_VAR
Serializer.AddTod(activeData);
END_METHOD

PROPERTY PUBLIC Size : UDINT
GET
Size := SIZEOF(activeData);
END_GET
END_PROPERTY

METHOD TryDeserializeFrom : BOOL
VAR_INPUT
	Deserializer : I_Deserializer;
	Feedback : I_DeserializerFeedback;
END_VAR
TryDeserializeFrom := Deserializer.TryGetTod(activeData, Feedback);
END_METHOD

METHOD TryMakeReferenceTo : BOOL
VAR_INPUT
	Target : I_Datatype;
END_VAR
VAR
	pTargetData : POINTER TO TIME_OF_DAY;
END_VAR
IF NOT (Target.TypeName = TypeName) THEN
	RETURN;
END_IF

pTargetData := Target.Address;
activeData REF= pTargetData^;
TryMakeReferenceTo := TRUE;
END_METHOD

PROPERTY PUBLIC TypeName : T_MAXSTRING
GET
TypeName := 'TIME_OF_DAY';
END_GET
END_PROPERTY

PROPERTY PUBLIC Value : TIME_OF_DAY
GET
Value := activeData;
END_GET
SET
activeData := Value;
END_SET
END_PROPERTY

END_FUNCTION_BLOCK

// Primitive/_TOD
{attribute 'linkalways'} 
{attribute 'no_explicit_call' := 'This FB is a CLASS and must be accessed using methods or properties'}
{attribute 'enable_dynamic_creation'}
FUNCTION_BLOCK _TOD EXTENDS DatatypeBase
VAR
	localData : TOD;
	activeData : REFERENCE TO TOD REF= localData;
END_VAR

METHOD FB_init : BOOL
VAR_INPUT
	bInitRetains : BOOL; // if TRUE, the retain variables are initialized (warm start / cold start)
	bInCopyCode : BOOL;  // if TRUE, the instance afterwards gets moved WORDo the copy code (online change)
	InitialValue : TOD;
END_VAR
localData := InitialValue;
END_METHOD

PROPERTY PUBLIC Address : PVOID
GET
Address := ADR(activeData);
END_GET
END_PROPERTY

METHOD PUBLIC ClearReference
VAR_INPUT
END_VAR
activeData REF= localData;
END_METHOD

METHOD PUBLIC Clone : I_Datatype
VAR
    pClone : POINTER TO _TOD;
END_VAR
pClone := __NEW(_TOD(InitialValue := Value));
Clone := pClone^;
END_METHOD

METHOD PUBLIC MakeReferenceTo
VAR_INPUT
	ReferenceTarget : REFERENCE TO TOD;
END_VAR
activeData REF= ReferenceTarget;
END_METHOD

METHOD PUBLIC SerializeWith
VAR_INPUT
	Serializer : I_Serializer;
END_VAR
Serializer.AddTod(activeData);
END_METHOD

PROPERTY PUBLIC Size : UDINT
GET
Size := SIZEOF(activeData);
END_GET
END_PROPERTY

METHOD TryDeserializeFrom : BOOL
VAR_INPUT
	Deserializer : I_Deserializer;
	Feedback : I_DeserializerFeedback;
END_VAR
TryDeserializeFrom := Deserializer.TryGetTod(activeData, Feedback);
END_METHOD

METHOD TryMakeReferenceTo : BOOL
VAR_INPUT
	Target : I_Datatype;
END_VAR
VAR
	pTargetData : POINTER TO TOD;
END_VAR
IF NOT (Target.TypeName = TypeName) THEN
	RETURN;
END_IF

pTargetData := Target.Address;
activeData REF= pTargetData^;
TryMakeReferenceTo := TRUE;
END_METHOD

PROPERTY PUBLIC TypeName : T_MAXSTRING
GET
TypeName := 'TOD';
END_GET
END_PROPERTY

PROPERTY PUBLIC Value : TOD
GET
Value := activeData;
END_GET
SET
activeData := Value;
END_SET
END_PROPERTY

END_FUNCTION_BLOCK

// Primitive/_UDINT
{attribute 'linkalways'} 
{attribute 'no_explicit_call' := 'This FB is a CLASS and must be accessed using methods or properties'}
{attribute 'enable_dynamic_creation'}
FUNCTION_BLOCK _UDINT EXTENDS NumericDatatypeBase
VAR
	localData : UDINT;
	activeData : REFERENCE TO UDINT REF= localData;
END_VAR

METHOD FB_init : BOOL
VAR_INPUT
	bInitRetains : BOOL; // if TRUE, the retain variables are initialized (warm start / cold start)
	bInCopyCode : BOOL;  // if TRUE, the instance afterwards gets moved into the copy code (online change)
	InitialValue : UDINT;
END_VAR
localData := InitialValue;
END_METHOD

METHOD PROTECTED SerializeMaxValue
VAR_INPUT
	Serializer : I_Serializer;
END_VAR
Serializer.AddUdint(MaxValue);
END_METHOD

METHOD PROTECTED SerializeMinValue
VAR_INPUT
	Serializer : I_Serializer;
END_VAR
Serializer.AddUdint(MinValue);
END_METHOD

PROPERTY PUBLIC Address : PVOID
GET
Address := ADR(activeData);
END_GET
END_PROPERTY

METHOD PUBLIC ClearReference
VAR_INPUT
END_VAR
activeData REF= localData;
END_METHOD

METHOD PUBLIC Clone : I_Datatype
VAR
    pClone : POINTER TO _UDINT;
END_VAR
pClone := __NEW(_UDINT(InitialValue := Value));
Clone := pClone^;
END_METHOD

PROPERTY PUBLIC IsFloat : BOOL
GET
IsFloat := FALSE;
END_GET
END_PROPERTY

PROPERTY PUBLIC IsSigned : BOOL
GET
IsSigned := FALSE;
END_GET
END_PROPERTY

METHOD PUBLIC MakeReferenceTo
VAR_INPUT
	ReferenceTarget : REFERENCE TO UDINT;
END_VAR
activeData REF= ReferenceTarget;
END_METHOD

PROPERTY PUBLIC MaxValue : UDINT
GET
MaxValue :=  DatatypeLimits.UDINT_MAX_VALUE;
END_GET
END_PROPERTY

PROPERTY PUBLIC MinValue : UDINT
GET
MinValue := DatatypeLimits.UDINT_MIN_VALUE;
END_GET
END_PROPERTY

METHOD PUBLIC SerializeWith
VAR_INPUT
	Serializer : I_Serializer;
END_VAR
Serializer.AddUdint(activeData);
END_METHOD

PROPERTY PUBLIC Size : UDINT
GET
Size := SIZEOF(activeData);
END_GET
END_PROPERTY

METHOD TryDeserializeFrom : BOOL
VAR_INPUT
	Deserializer : I_Deserializer;
	Feedback : I_DeserializerFeedback;
END_VAR
TryDeserializeFrom := Deserializer.TryGetUdint(activeData, Feedback);
END_METHOD

METHOD TryMakeReferenceTo : BOOL
VAR_INPUT
	Target : I_Datatype;
END_VAR
VAR
	pTargetData : POINTER TO UDINT;
END_VAR
IF NOT (Target.TypeName = TypeName) THEN
	RETURN;
END_IF

pTargetData := Target.Address;
activeData REF= pTargetData^;
TryMakeReferenceTo := TRUE;
END_METHOD

PROPERTY PUBLIC TypeName : T_MAXSTRING
GET
TypeName := 'UDINT';
END_GET
END_PROPERTY

PROPERTY PUBLIC Value : UDINT
GET
Value := activeData;
END_GET
SET
activeData := Value;
END_SET
END_PROPERTY

END_FUNCTION_BLOCK

// Primitive/_UINT
{attribute 'linkalways'} 
{attribute 'no_explicit_call' := 'This FB is a CLASS and must be accessed using methods or properties'}
{attribute 'enable_dynamic_creation'}
FUNCTION_BLOCK _UINT EXTENDS NumericDatatypeBase
VAR
	localData : UINT;
	activeData : REFERENCE TO UINT REF= localData;
END_VAR

METHOD FB_init : BOOL
VAR_INPUT
	bInitRetains : BOOL; // if TRUE, the retain variables are initialized (warm start / cold start)
	bInCopyCode : BOOL;  // if TRUE, the instance afterwards gets moved into the copy code (online change)
	InitialValue : UINT;
END_VAR
localData := InitialValue;
END_METHOD

METHOD PROTECTED SerializeMaxValue
VAR_INPUT
	Serializer : I_Serializer;
END_VAR
Serializer.AddUint(MaxValue);
END_METHOD

METHOD PROTECTED SerializeMinValue
VAR_INPUT
	Serializer : I_Serializer;
END_VAR
Serializer.AddUint(MinValue);
END_METHOD

PROPERTY PUBLIC Address : PVOID
GET
Address := ADR(activeData);
END_GET
END_PROPERTY

METHOD PUBLIC ClearReference
VAR_INPUT
END_VAR
activeData REF= localData;
END_METHOD

METHOD PUBLIC Clone : I_Datatype
VAR
    pClone : POINTER TO _UINT;
END_VAR
pClone := __NEW(_UINT(InitialValue := Value));
Clone := pClone^;
END_METHOD

PROPERTY PUBLIC IsFloat : BOOL
GET
IsFloat := FALSE;
END_GET
END_PROPERTY

PROPERTY PUBLIC IsSigned : BOOL
GET
IsSigned := FALSE;
END_GET
END_PROPERTY

METHOD PUBLIC MakeReferenceTo
VAR_INPUT
	ReferenceTarget : REFERENCE TO UINT;
END_VAR
activeData REF= ReferenceTarget;
END_METHOD

PROPERTY PUBLIC MaxValue : UINT
GET
MaxValue :=  DatatypeLimits.UINT_MAX_VALUE;
END_GET
END_PROPERTY

PROPERTY PUBLIC MinValue : UINT
GET
MinValue := DatatypeLimits.UINT_MIN_VALUE;
END_GET
END_PROPERTY

METHOD PUBLIC SerializeWith
VAR_INPUT
	Serializer : I_Serializer;
END_VAR
Serializer.AddUint(activeData);
END_METHOD

PROPERTY PUBLIC Size : UDINT
GET
Size := SIZEOF(activeData);
END_GET
END_PROPERTY

METHOD TryDeserializeFrom : BOOL
VAR_INPUT
	Deserializer : I_Deserializer;
	Feedback : I_DeserializerFeedback;
END_VAR
TryDeserializeFrom := Deserializer.TryGetUint(activeData, Feedback);
END_METHOD

METHOD TryMakeReferenceTo : BOOL
VAR_INPUT
	Target : I_Datatype;
END_VAR
VAR
	pTargetData : POINTER TO UINT;
END_VAR
IF NOT (Target.TypeName = TypeName) THEN
	RETURN;
END_IF

pTargetData := Target.Address;
activeData REF= pTargetData^;
TryMakeReferenceTo := TRUE;
END_METHOD

PROPERTY PUBLIC TypeName : T_MAXSTRING
GET
TypeName := 'UINT';
END_GET
END_PROPERTY

PROPERTY PUBLIC Value : UINT
GET
Value := activeData;
END_GET
SET
activeData := Value;
END_SET
END_PROPERTY

END_FUNCTION_BLOCK

// Primitive/_ULINT
{attribute 'linkalways'} 
{attribute 'no_explicit_call' := 'This FB is a CLASS and must be accessed using methods or properties'}
{attribute 'enable_dynamic_creation'}
FUNCTION_BLOCK _ULINT EXTENDS NumericDatatypeBase
VAR
	localData : ULINT;
	activeData : REFERENCE TO ULINT REF= localData;
END_VAR

METHOD FB_init : BOOL
VAR_INPUT
	bInitRetains : BOOL; // if TRUE, the retain variables are initialized (warm start / cold start)
	bInCopyCode : BOOL;  // if TRUE, the instance afterwards gets moved into the copy code (online change)
	InitialValue : ULINT;
END_VAR
localData := InitialValue;
END_METHOD

METHOD PROTECTED SerializeMaxValue
VAR_INPUT
	Serializer : I_Serializer;
END_VAR
Serializer.AddUlint(MaxValue);
END_METHOD

METHOD PROTECTED SerializeMinValue
VAR_INPUT
	Serializer : I_Serializer;
END_VAR
Serializer.AddUlint(MinValue);
END_METHOD

PROPERTY PUBLIC Address : PVOID
GET
Address := ADR(activeData);
END_GET
END_PROPERTY

METHOD PUBLIC ClearReference
VAR_INPUT
END_VAR
activeData REF= localData;
END_METHOD

METHOD PUBLIC Clone : I_Datatype
VAR
    pClone : POINTER TO _ULINT;
END_VAR
pClone := __NEW(_ULINT(InitialValue := Value));
Clone := pClone^;
END_METHOD

PROPERTY PUBLIC IsFloat : BOOL
GET
IsFloat := FALSE;
END_GET
END_PROPERTY

PROPERTY PUBLIC IsSigned : BOOL
GET
IsSigned := FALSE;
END_GET
END_PROPERTY

METHOD PUBLIC MakeReferenceTo
VAR_INPUT
	ReferenceTarget : REFERENCE TO ULINT;
END_VAR
activeData REF= ReferenceTarget;
END_METHOD

PROPERTY PUBLIC MaxValue : ULINT
GET
MaxValue :=  DatatypeLimits.ULINT_MAX_VALUE;
END_GET
END_PROPERTY

PROPERTY PUBLIC MinValue : ULINT
GET
MinValue := DatatypeLimits.ULINT_MIN_VALUE;
END_GET
END_PROPERTY

METHOD PUBLIC SerializeWith
VAR_INPUT
	Serializer : I_Serializer;
END_VAR
Serializer.AddUlint(activeData);
END_METHOD

PROPERTY PUBLIC Size : UDINT
GET
Size := SIZEOF(activeData);
END_GET
END_PROPERTY

METHOD TryDeserializeFrom : BOOL
VAR_INPUT
	Deserializer : I_Deserializer;
	Feedback : I_DeserializerFeedback;
END_VAR
TryDeserializeFrom := Deserializer.TryGetUlint(activeData, Feedback);
END_METHOD

METHOD TryMakeReferenceTo : BOOL
VAR_INPUT
	Target : I_Datatype;
END_VAR
VAR
	pTargetData : POINTER TO ULINT;
END_VAR
IF NOT (Target.TypeName = TypeName) THEN
	RETURN;
END_IF

pTargetData := Target.Address;
activeData REF= pTargetData^;
TryMakeReferenceTo := TRUE;
END_METHOD

PROPERTY PUBLIC TypeName : T_MAXSTRING
GET
TypeName := 'ULINT';
END_GET
END_PROPERTY

PROPERTY PUBLIC Value : ULINT
GET
Value := activeData;
END_GET
SET
activeData := Value;
END_SET
END_PROPERTY

END_FUNCTION_BLOCK

// Primitive/_USINT
{attribute 'linkalways'} 
{attribute 'no_explicit_call' := 'This FB is a CLASS and must be accessed using methods or properties'}
{attribute 'enable_dynamic_creation'}
FUNCTION_BLOCK _USINT EXTENDS NumericDatatypeBase
VAR
	localData : USINT;
	activeData : REFERENCE TO USINT REF= localData;
END_VAR

METHOD FB_init : BOOL
VAR_INPUT
	bInitRetains : BOOL; // if TRUE, the retain variables are initialized (warm start / cold start)
	bInCopyCode : BOOL;  // if TRUE, the instance afterwards gets moved into the copy code (online change)
	InitialValue : USINT;
END_VAR
localData := InitialValue;
END_METHOD

METHOD PROTECTED SerializeMaxValue
VAR_INPUT
	Serializer : I_Serializer;
END_VAR
Serializer.AddUsint(MaxValue);
END_METHOD

METHOD PROTECTED SerializeMinValue
VAR_INPUT
	Serializer : I_Serializer;
END_VAR
Serializer.AddUsint(MinValue);
END_METHOD

PROPERTY PUBLIC Address : PVOID
GET
Address := ADR(activeData);
END_GET
END_PROPERTY

METHOD PUBLIC ClearReference
VAR_INPUT
END_VAR
activeData REF= localData;
END_METHOD

METHOD PUBLIC Clone : I_Datatype
VAR
    pClone : POINTER TO _USINT;
END_VAR
pClone := __NEW(_USINT(InitialValue := Value));
Clone := pClone^;
END_METHOD

PROPERTY PUBLIC IsFloat : BOOL
GET
IsFloat := FALSE;
END_GET
END_PROPERTY

PROPERTY PUBLIC IsSigned : BOOL
GET
IsSigned := FALSE;
END_GET
END_PROPERTY

METHOD PUBLIC MakeReferenceTo
VAR_INPUT
	ReferenceTarget : REFERENCE TO USINT;
END_VAR
activeData REF= ReferenceTarget;
END_METHOD

PROPERTY PUBLIC MaxValue : USINT
GET
MaxValue :=  DatatypeLimits.USINT_MAX_VALUE;
END_GET
END_PROPERTY

PROPERTY PUBLIC MinValue : USINT
GET
MinValue := DatatypeLimits.USINT_MIN_VALUE;
END_GET
END_PROPERTY

METHOD PUBLIC SerializeWith
VAR_INPUT
	Serializer : I_Serializer;
END_VAR
Serializer.AddUsint(activeData);
END_METHOD

PROPERTY PUBLIC Size : UDINT
GET
Size := SIZEOF(activeData);
END_GET
END_PROPERTY

METHOD TryDeserializeFrom : BOOL
VAR_INPUT
	Deserializer : I_Deserializer;
	Feedback : I_DeserializerFeedback;
END_VAR
TryDeserializeFrom := Deserializer.TryGetUsint(activeData, Feedback);
END_METHOD

METHOD TryMakeReferenceTo : BOOL
VAR_INPUT
	Target : I_Datatype;
END_VAR
VAR
	pTargetData : POINTER TO USINT;
END_VAR
IF NOT (Target.TypeName = TypeName) THEN
	RETURN;
END_IF

pTargetData := Target.Address;
activeData REF= pTargetData^;
TryMakeReferenceTo := TRUE;
END_METHOD

PROPERTY PUBLIC TypeName : T_MAXSTRING
GET
TypeName := 'USINT';
END_GET
END_PROPERTY

PROPERTY PUBLIC Value : USINT
GET
Value := activeData;
END_GET
SET
activeData := Value;
END_SET
END_PROPERTY

END_FUNCTION_BLOCK

// Primitive/_WORD
{attribute 'linkalways'} 
{attribute 'no_explicit_call' := 'This FB is a CLASS and must be accessed using methods or properties'}
{attribute 'enable_dynamic_creation'}
FUNCTION_BLOCK _WORD EXTENDS NumericDatatypeBase
VAR
	localData : WORD;
	activeData : REFERENCE TO WORD REF= localData;
END_VAR

METHOD FB_init : BOOL
VAR_INPUT
	bInitRetains : BOOL; // if TRUE, the retain variables are initialized (warm start / cold start)
	bInCopyCode : BOOL;  // if TRUE, the instance afterwards gets moved WORDo the copy code (online change)
	InitialValue : WORD;
END_VAR
localData := InitialValue;
END_METHOD

METHOD PROTECTED SerializeMaxValue
VAR_INPUT
	Serializer : I_Serializer;
END_VAR
Serializer.AddWord(MaxValue);
END_METHOD

METHOD PROTECTED SerializeMinValue
VAR_INPUT
	Serializer : I_Serializer;
END_VAR
Serializer.AddWord(MinValue);
END_METHOD

PROPERTY PUBLIC Address : PVOID
GET
Address := ADR(activeData);
END_GET
END_PROPERTY

METHOD PUBLIC ClearReference
VAR_INPUT
END_VAR
activeData REF= localData;
END_METHOD

METHOD PUBLIC Clone : I_Datatype
VAR
    pClone : POINTER TO _WORD;
END_VAR
pClone := __NEW(_WORD(InitialValue := Value));
Clone := pClone^;
END_METHOD

PROPERTY PUBLIC IsFloat : BOOL
GET
IsFloat := FALSE;
END_GET
END_PROPERTY

PROPERTY PUBLIC IsSigned : BOOL
GET
IsSigned := FALSE;
END_GET
END_PROPERTY

METHOD PUBLIC MakeReferenceTo
VAR_INPUT
	ReferenceTarget : REFERENCE TO WORD;
END_VAR
activeData REF= ReferenceTarget;
END_METHOD

PROPERTY PUBLIC MaxValue : WORD
GET
MaxValue :=  DatatypeLimits.WORD_MAX_VALUE;
END_GET
END_PROPERTY

PROPERTY PUBLIC MinValue : WORD
GET
MinValue := DatatypeLimits.WORD_MIN_VALUE;
END_GET
END_PROPERTY

METHOD PUBLIC SerializeWith
VAR_INPUT
	Serializer : I_Serializer;
END_VAR
Serializer.AddWord(activeData);
END_METHOD

PROPERTY PUBLIC Size : UDINT
GET
Size := SIZEOF(activeData);
END_GET
END_PROPERTY

METHOD TryDeserializeFrom : BOOL
VAR_INPUT
	Deserializer : I_Deserializer;
	Feedback : I_DeserializerFeedback;
END_VAR
TryDeserializeFrom := Deserializer.TryGetWord(activeData, Feedback);
END_METHOD

METHOD TryMakeReferenceTo : BOOL
VAR_INPUT
	Target : I_Datatype;
END_VAR
VAR
	pTargetData : POINTER TO WORD;
END_VAR
IF NOT (Target.TypeName = TypeName) THEN
	RETURN;
END_IF

pTargetData := Target.Address;
activeData REF= pTargetData^;
TryMakeReferenceTo := TRUE;
END_METHOD

PROPERTY PUBLIC TypeName : T_MAXSTRING
GET
TypeName := 'WORD';
END_GET
END_PROPERTY

PROPERTY PUBLIC Value : WORD
GET
Value := activeData;
END_GET
SET
activeData := Value;
END_SET
END_PROPERTY

END_FUNCTION_BLOCK

// PrimitiveDatatypePack
{attribute 'linkalways'} 
{attribute 'no_explicit_call' := 'This FB is a CLASS and must be accessed using methods or properties'}
{attribute 'enable_dynamic_creation'}
FUNCTION_BLOCK PrimitiveDatatypePack IMPLEMENTS I_DatatypePack
VAR
	
	_bool : _BOOL(FALSE);
	_byte : _BYTE(0);
	_dint : _DINT(0);
	_dt : _DT(DT#1970-1-1-0:0:0);
	_dword : _DWORD(0);
	_int : _INT(0);
	_lint : _LINT(0);
	_lreal : _LREAL(0);
	_lword : _LWORD(0);
	_real : _REAL(0);
	_sint : _SINT(0);
	_time_of_day : _TIME_OF_DAY(TOD#0:0:0);
	_tod : _TOD(TOD#0:0:0);
	_udint : _UDINT(0);
	_uint : _UINT(0);
	_ulint : _ULINT(0);
	_usint : _USINT(0);
	_word : _WORD(0);
    _string : _STRING('');
	
END_VAR

METHOD RegisterWith
VAR_INPUT
	Datatypes : I_Datatypes;
END_VAR
Datatypes.RegisterDatatype(_bool);
Datatypes.RegisterDatatype(_byte);
Datatypes.RegisterDatatype(_dint);
Datatypes.RegisterDatatype(_dt);
Datatypes.RegisterDatatype(_dword);
Datatypes.RegisterDatatype(_int);
Datatypes.RegisterDatatype(_lint);
Datatypes.RegisterDatatype(_lreal);
Datatypes.RegisterDatatype(_lword);
Datatypes.RegisterDatatype(_real);
Datatypes.RegisterDatatype(_sint);
Datatypes.RegisterDatatype(_time_of_day);
Datatypes.RegisterDatatype(_tod);
Datatypes.RegisterDatatype(_udint);
Datatypes.RegisterDatatype(_uint);
Datatypes.RegisterDatatype(_ulint);
Datatypes.RegisterDatatype(_usint);
Datatypes.RegisterDatatype(_word);
Datatypes.RegisterDatatype(_string);
END_METHOD

END_FUNCTION_BLOCK
